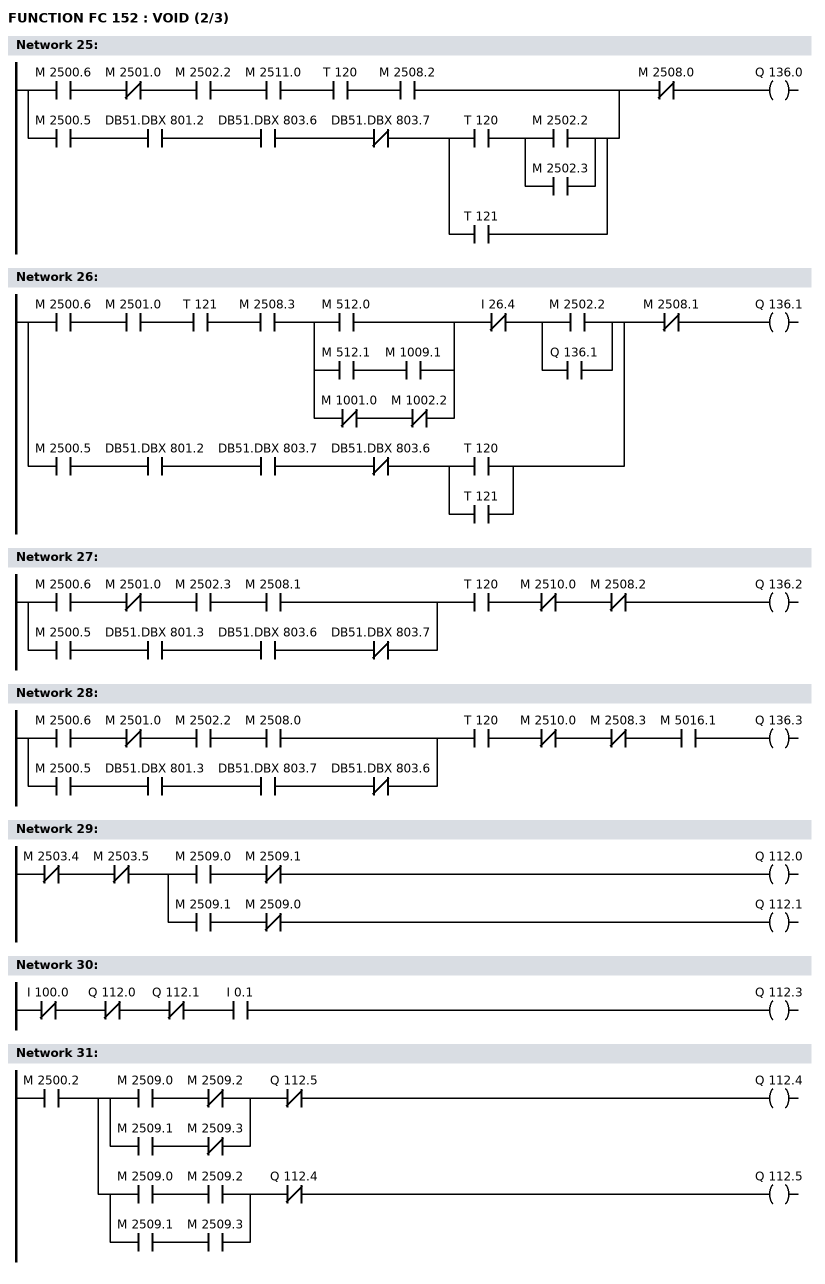

      A(    ;
      A     M   2500.6;
      AN    M   2501.0;
      A     M   2502.2;
      A     M   2511.0;
      A     T    120;
      A     M   2508.2;
      O     ;
      A     M   2500.5;
      A     DB51.DBX  801.2;
      A     DB51.DBX  803.6;
      AN    DB51.DBX  803.7;
      A(    ;
      A     T    120;
      A(    ;
      O     M   2502.2;
      O     M   2502.3;
      )     ;
      O     T    121;
      )     ;
      )     ;
      AN    M   2508.0;
      =     Q    136.0;
NETWORK
TITLE =

      A(    ;
      A     M   2500.6;
      A     M   2501.0;
      A     T    121;
      A     M   2508.3;
      A(    ;
      O     M    512.0;
      O     ;
      A     M    512.1;
      A     M   1009.1;
      O     ;
      AN    M   1001.0;
      AN    M   1002.2;
      )     ;
      AN    I     26.4;
      A(    ;
      O     M   2502.2;
      O     Q    136.1;
      )     ;
      O     ;
      A     M   2500.5;
      A     DB51.DBX  801.2;
      A     DB51.DBX  803.7;
      AN    DB51.DBX  803.6;
      A(    ;
      O     T    120;
      O     T    121;
      )     ;
      )     ;
      AN    M   2508.1;
      =     Q    136.1;
NETWORK
TITLE =

      A(    ;
      A     M   2500.6;
      AN    M   2501.0;
      A     M   2502.3;
      A     M   2508.1;
      O     ;
      A     M   2500.5;
      A     DB51.DBX  801.3;
      A     DB51.DBX  803.6;
      AN    DB51.DBX  803.7;
      )     ;
      A     T    120;
      AN    M   2510.0;
      AN    M   2508.2;
      =     Q    136.2;
NETWORK
TITLE =

      A(    ;
      A     M   2500.6;
      AN    M   2501.0;
      A     M   2502.2;
      A     M   2508.0;
      O     ;
      A     M   2500.5;
      A     DB51.DBX  801.3;
      A     DB51.DBX  803.7;
      AN    DB51.DBX  803.6;
      )     ;
      A     T    120;
      AN    M   2510.0;
      AN    M   2508.3;
      A     M   5016.1;
      =     Q    136.3;
NETWORK
TITLE =

      AN    M   2503.4;
      AN    M   2503.5;
      =     L      0.0;
      A     L      0.0;
      A     M   2509.0;
      AN    M   2509.1;
      =     Q    112.0;
      A     L      0.0;
      A     M   2509.1;
      AN    M   2509.0;
      =     Q    112.1;
NETWORK
TITLE =

      AN    I    100.0;
      AN    Q    112.0;
      AN    Q    112.1;
      A     I      0.1;
      =     Q    112.3;
NETWORK
TITLE =

      A     M   2500.2;
      =     L      0.0;
      A     L      0.0;
      A(    ;
      A     M   2509.0;
      AN    M   2509.2;
      O     ;
      A     M   2509.1;
      AN    M   2509.3;
      )     ;
      AN    Q    112.5;
      =     Q    112.4;
      A     L      0.0;
      A(    ;
      A     M   2509.0;
      A     M   2509.2;
      O     ;
      A     M   2509.1;
      A     M   2509.3;
      )     ;
      AN    Q    112.4;
      =     Q    112.5;
NETWORK
TITLE =
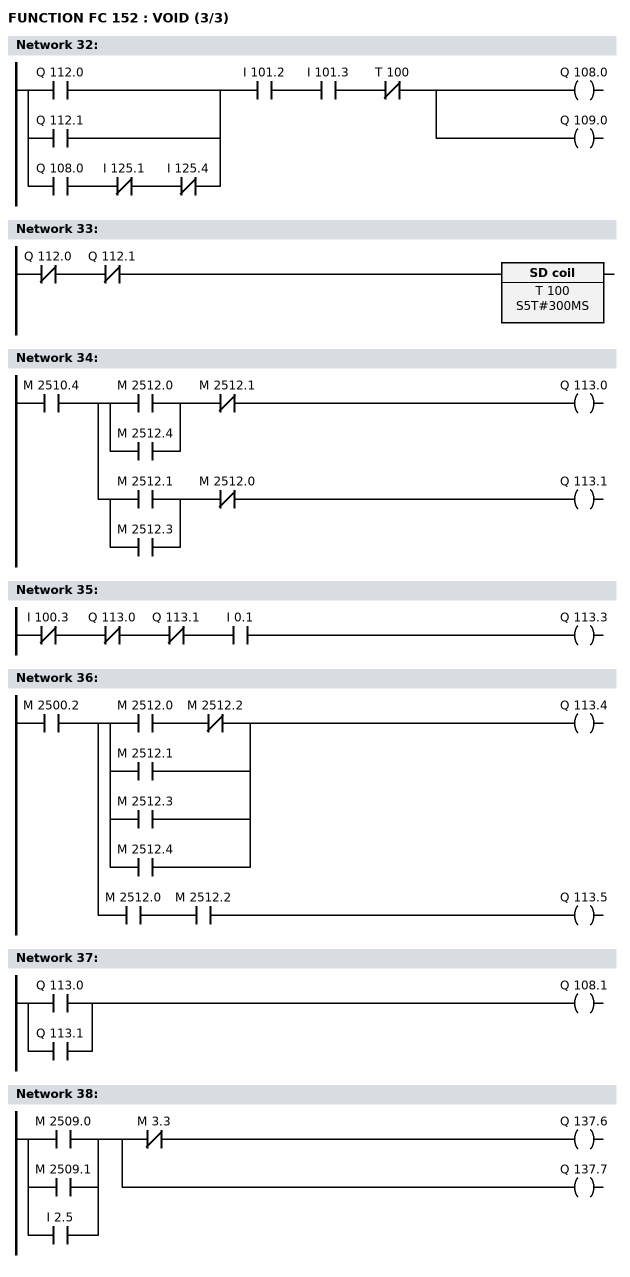

      A(    ;
      O     Q    112.0;
      O     Q    112.1;
      O     ;
      A     Q    108.0;
      AN    I    125.1;
      AN    I    125.4;
      )     ;
      A     I    101.2;
      A     I    101.3;
      AN    T    100;
      =     Q    108.0;
      =     Q    109.0;
NETWORK
TITLE =

      AN    Q    112.0;
      AN    Q    112.1;
      L     S5T#300MS;
      SD    T    100;
NETWORK
TITLE =

      A     M   2510.4;
      =     L      0.0;
      A     L      0.0;
      A(    ;
      O     M   2512.0;
      O     M   2512.4;
      )     ;
      AN    M   2512.1;
      =     Q    113.0;
      A     L      0.0;
      A(    ;
      O     M   2512.1;
      O     M   2512.3;
      )     ;
      AN    M   2512.0;
      =     Q    113.1;
NETWORK
TITLE =

      AN    I    100.3;
      AN    Q    113.0;
      AN    Q    113.1;
      A     I      0.1;
      =     Q    113.3;
NETWORK
TITLE =

      A     M   2500.2;
      =     L      0.0;
      A     L      0.0;
      A(    ;
      A     M   2512.0;
      AN    M   2512.2;
      O     M   2512.1;
      O     M   2512.3;
      O     M   2512.4;
      )     ;
      =     Q    113.4;
      A     L      0.0;
      A     M   2512.0;
      A     M   2512.2;
      =     Q    113.5;
NETWORK
TITLE =

      O     Q    113.0;
      O     Q    113.1;
      =     Q    108.1;
NETWORK
TITLE =

      O     M   2509.0;
      O     M   2509.1;
      O     I      2.5;
      =     L      0.0;
      A     L      0.0;
      AN    M      3.3;
      =     Q    137.6;
      A     L      0.0;
      BLD   102;
      =     Q    137.7;
END_FUNCTION

FUNCTION FC 324 : VOID
TITLE =
VERSION : 0.1

BEGIN
NETWORK
TITLE =DP DIAGNOSTIC FOR DP MASTER SYSTEM(1)

      AN    OV;
      =     L      0.0;
      BLD   103;
      A     OV;
      =     L      0.1;
      BLD   103;
      CALL FC   325 (
           CHECK_ACTIV              := L      0.0,
           EXTERNAL_DP_INTERFACE    := L      0.1,
           DP_MASTERSYSTEM          := 1,
           DATA_FIELD               := P#DB325.DBX0.0 BYTE 50,
           SUM_SLAVES_DIAG          := DB325.DBW   82,
           LIST_SLAVES_NOT_PRESENT  := P#DB325.DBX 50.0 DWORD 4,
           LIST_SLAVES_ERROR        := P#DB325.DBX 66.0 DWORD 4,
           RETVAL                   := DB325.DBW   84,
           BUSY                     := DB325.DBX   90.0);
      NOP   0;
NETWORK
TITLE =#702R1
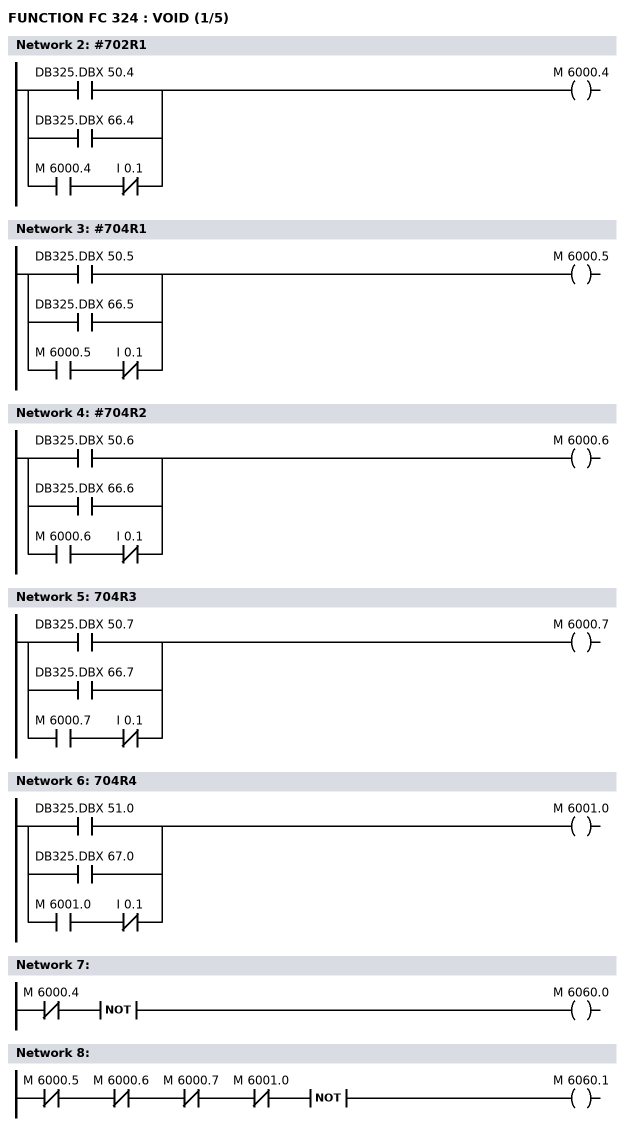

      O     DB325.DBX   50.4;
      O     DB325.DBX   66.4;
      O     ;
      A     M   6000.4;
      AN    I      0.1;
      =     M   6000.4;
NETWORK
TITLE =#704R1

      O     DB325.DBX   50.5;
      O     DB325.DBX   66.5;
      O     ;
      A     M   6000.5;
      AN    I      0.1;
      =     M   6000.5;
NETWORK
TITLE =#704R2

      O     DB325.DBX   50.6;
      O     DB325.DBX   66.6;
      O     ;
      A     M   6000.6;
      AN    I      0.1;
      =     M   6000.6;
NETWORK
TITLE =704R3

      O     DB325.DBX   50.7;
      O     DB325.DBX   66.7;
      O     ;
      A     M   6000.7;
      AN    I      0.1;
      =     M   6000.7;
NETWORK
TITLE =704R4

      O     DB325.DBX   51.0;
      O     DB325.DBX   67.0;
      O     ;
      A     M   6001.0;
      AN    I      0.1;
      =     M   6001.0;
NETWORK
TITLE =

      AN    M   6000.4;
      NOT   ;
      =     M   6060.0;
NETWORK
TITLE =

      AN    M   6000.5;
      AN    M   6000.6;
      AN    M   6000.7;
      AN    M   6001.0;
      NOT   ;
      =     M   6060.1;
NETWORK
TITLE =
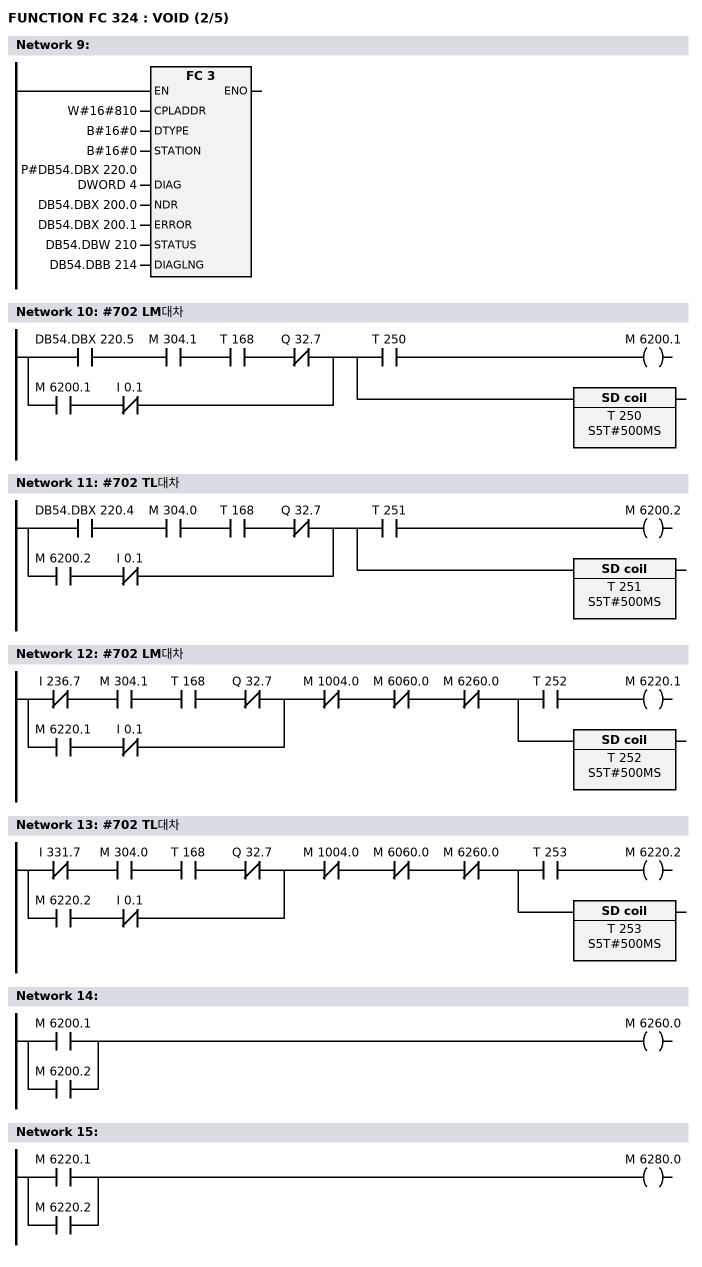

      CALL FC     3 (
           CPLADDR                  := W#16#810,
           DTYPE                    := B#16#0,
           STATION                  := B#16#0,
           DIAG                     := P#DB54.DBX 220.0 DWORD 4,
           NDR                      := DB54.DBX  200.0,
           ERROR                    := DB54.DBX  200.1,
           STATUS                   := DB54.DBW  210,
           DIAGLNG                  := DB54.DBB  214);
      NOP   0;
NETWORK
TITLE =#702 LM대차

      A     DB54.DBX  220.5;
      A     M    304.1;
      A     T    168;
      AN    Q     32.7;
      O     ;
      A     M   6200.1;
      AN    I      0.1;
      =     L      0.0;
      A     L      0.0;
      A     T    250;
      =     M   6200.1;
      A     L      0.0;
      BLD   102;
      L     S5T#500MS;
      SD    T    250;
NETWORK
TITLE =#702 TL대차

      A     DB54.DBX  220.4;
      A     M    304.0;
      A     T    168;
      AN    Q     32.7;
      O     ;
      A     M   6200.2;
      AN    I      0.1;
      =     L      0.0;
      A     L      0.0;
      A     T    251;
      =     M   6200.2;
      A     L      0.0;
      BLD   102;
      L     S5T#500MS;
      SD    T    251;
NETWORK
TITLE =#702 LM대차

      A(    ;
      AN    I    236.7;
      A     M    304.1;
      A     T    168;
      AN    Q     32.7;
      O     ;
      A     M   6220.1;
      AN    I      0.1;
      )     ;
      AN    M   1004.0;
      AN    M   6060.0;
      AN    M   6260.0;
      =     L      0.0;
      A     L      0.0;
      A     T    252;
      =     M   6220.1;
      A     L      0.0;
      BLD   102;
      L     S5T#500MS;
      SD    T    252;
NETWORK
TITLE =#702 TL대차

      A(    ;
      AN    I    331.7;
      A     M    304.0;
      A     T    168;
      AN    Q     32.7;
      O     ;
      A     M   6220.2;
      AN    I      0.1;
      )     ;
      AN    M   1004.0;
      AN    M   6060.0;
      AN    M   6260.0;
      =     L      0.0;
      A     L      0.0;
      A     T    253;
      =     M   6220.2;
      A     L      0.0;
      BLD   102;
      L     S5T#500MS;
      SD    T    253;
NETWORK
TITLE =

      O     M   6200.1;
      O     M   6200.2;
      =     M   6260.0;
NETWORK
TITLE =

      O     M   6220.1;
      O     M   6220.2;
      =     M   6280.0;
NETWORK
TITLE =
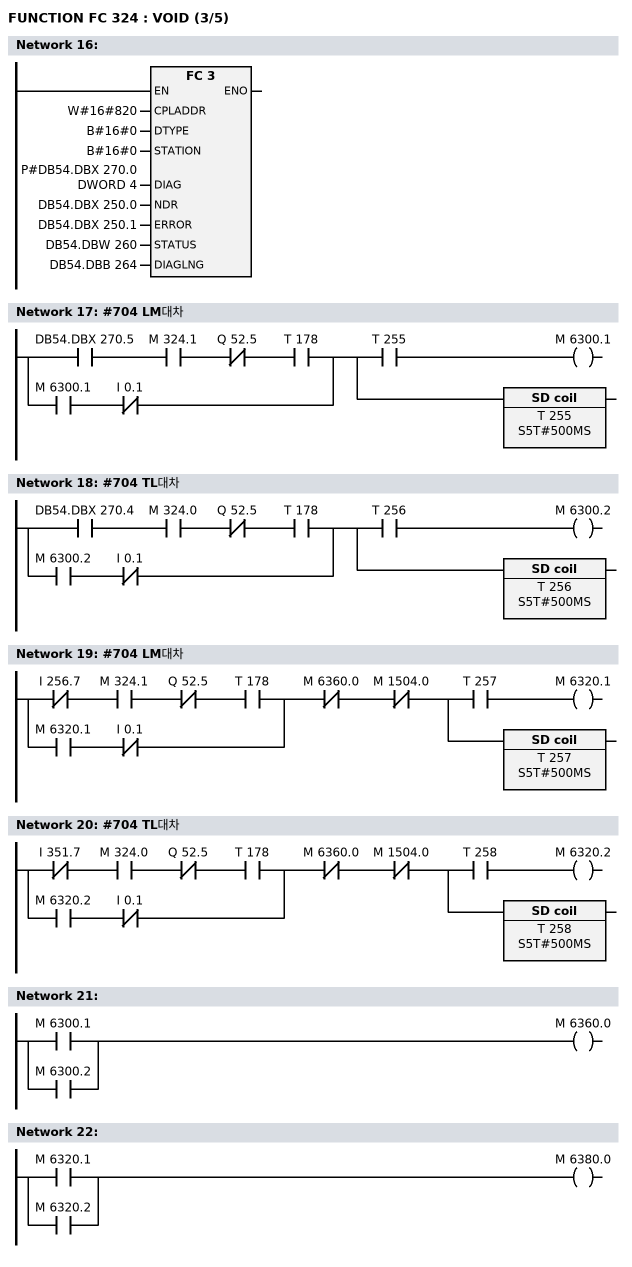

      CALL FC     3 (
           CPLADDR                  := W#16#820,
           DTYPE                    := B#16#0,
           STATION                  := B#16#0,
           DIAG                     := P#DB54.DBX 270.0 DWORD 4,
           NDR                      := DB54.DBX  250.0,
           ERROR                    := DB54.DBX  250.1,
           STATUS                   := DB54.DBW  260,
           DIAGLNG                  := DB54.DBB  264);
      NOP   0;
NETWORK
TITLE =#704 LM대차

      A     DB54.DBX  270.5;
      A     M    324.1;
      AN    Q     52.5;
      A     T    178;
      O     ;
      A     M   6300.1;
      AN    I      0.1;
      =     L      0.0;
      A     L      0.0;
      A     T    255;
      =     M   6300.1;
      A     L      0.0;
      BLD   102;
      L     S5T#500MS;
      SD    T    255;
NETWORK
TITLE =#704 TL대차

      A     DB54.DBX  270.4;
      A     M    324.0;
      AN    Q     52.5;
      A     T    178;
      O     ;
      A     M   6300.2;
      AN    I      0.1;
      =     L      0.0;
      A     L      0.0;
      A     T    256;
      =     M   6300.2;
      A     L      0.0;
      BLD   102;
      L     S5T#500MS;
      SD    T    256;
NETWORK
TITLE =#704 LM대차

      A(    ;
      AN    I    256.7;
      A     M    324.1;
      AN    Q     52.5;
      A     T    178;
      O     ;
      A     M   6320.1;
      AN    I      0.1;
      )     ;
      AN    M   6360.0;
      AN    M   1504.0;
      =     L      0.0;
      A     L      0.0;
      A     T    257;
      =     M   6320.1;
      A     L      0.0;
      BLD   102;
      L     S5T#500MS;
      SD    T    257;
NETWORK
TITLE =#704 TL대차

      A(    ;
      AN    I    351.7;
      A     M    324.0;
      AN    Q     52.5;
      A     T    178;
      O     ;
      A     M   6320.2;
      AN    I      0.1;
      )     ;
      AN    M   6360.0;
      AN    M   1504.0;
      =     L      0.0;
      A     L      0.0;
      A     T    258;
      =     M   6320.2;
      A     L      0.0;
      BLD   102;
      L     S5T#500MS;
      SD    T    258;
NETWORK
TITLE =

      O     M   6300.1;
      O     M   6300.2;
      =     M   6360.0;
NETWORK
TITLE =

      O     M   6320.1;
      O     M   6320.2;
      =     M   6380.0;
NETWORK
TITLE =
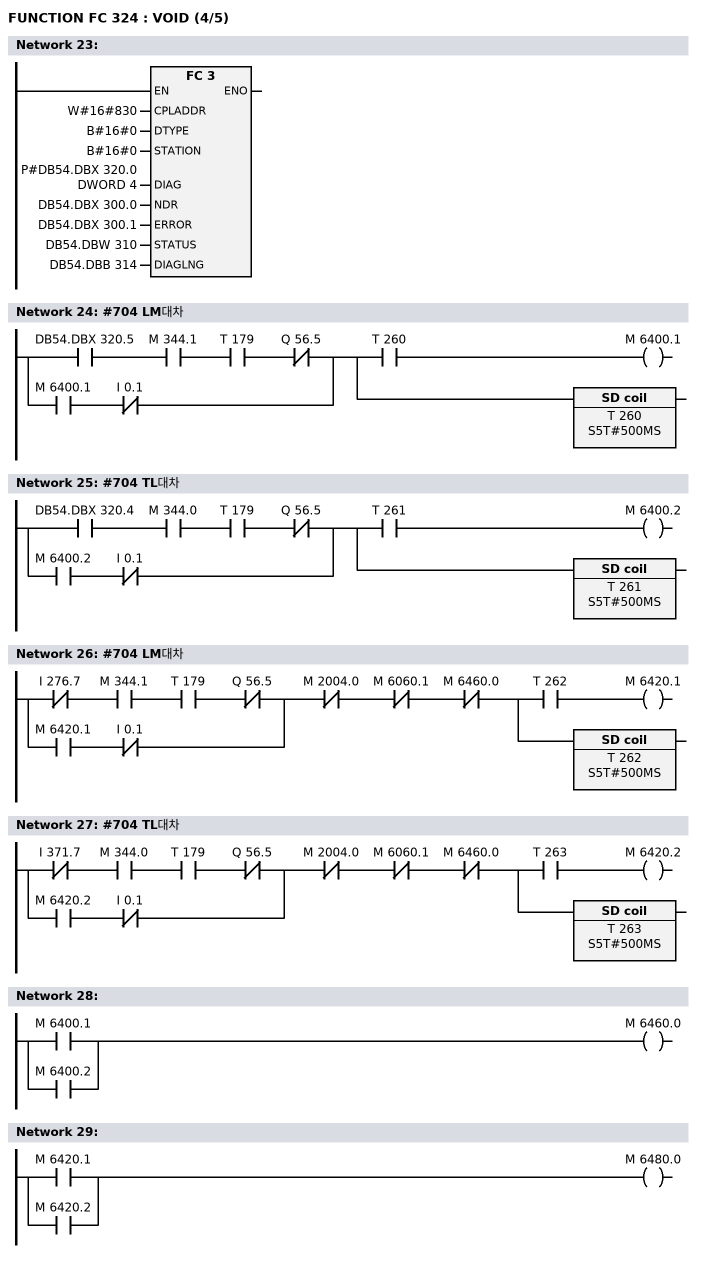

      CALL FC     3 (
           CPLADDR                  := W#16#830,
           DTYPE                    := B#16#0,
           STATION                  := B#16#0,
           DIAG                     := P#DB54.DBX 320.0 DWORD 4,
           NDR                      := DB54.DBX  300.0,
           ERROR                    := DB54.DBX  300.1,
           STATUS                   := DB54.DBW  310,
           DIAGLNG                  := DB54.DBB  314);
      NOP   0;
NETWORK
TITLE =#704 LM대차

      A     DB54.DBX  320.5;
      A     M    344.1;
      A     T    179;
      AN    Q     56.5;
      O     ;
      A     M   6400.1;
      AN    I      0.1;
      =     L      0.0;
      A     L      0.0;
      A     T    260;
      =     M   6400.1;
      A     L      0.0;
      BLD   102;
      L     S5T#500MS;
      SD    T    260;
NETWORK
TITLE =#704 TL대차

      A     DB54.DBX  320.4;
      A     M    344.0;
      A     T    179;
      AN    Q     56.5;
      O     ;
      A     M   6400.2;
      AN    I      0.1;
      =     L      0.0;
      A     L      0.0;
      A     T    261;
      =     M   6400.2;
      A     L      0.0;
      BLD   102;
      L     S5T#500MS;
      SD    T    261;
NETWORK
TITLE =#704 LM대차

      A(    ;
      AN    I    276.7;
      A     M    344.1;
      A     T    179;
      AN    Q     56.5;
      O     ;
      A     M   6420.1;
      AN    I      0.1;
      )     ;
      AN    M   2004.0;
      AN    M   6060.1;
      AN    M   6460.0;
      =     L      0.0;
      A     L      0.0;
      A     T    262;
      =     M   6420.1;
      A     L      0.0;
      BLD   102;
      L     S5T#500MS;
      SD    T    262;
NETWORK
TITLE =#704 TL대차

      A(    ;
      AN    I    371.7;
      A     M    344.0;
      A     T    179;
      AN    Q     56.5;
      O     ;
      A     M   6420.2;
      AN    I      0.1;
      )     ;
      AN    M   2004.0;
      AN    M   6060.1;
      AN    M   6460.0;
      =     L      0.0;
      A     L      0.0;
      A     T    263;
      =     M   6420.2;
      A     L      0.0;
      BLD   102;
      L     S5T#500MS;
      SD    T    263;
NETWORK
TITLE =

      O     M   6400.1;
      O     M   6400.2;
      =     M   6460.0;
NETWORK
TITLE =

      O     M   6420.1;
      O     M   6420.2;
      =     M   6480.0;
NETWORK
TITLE =
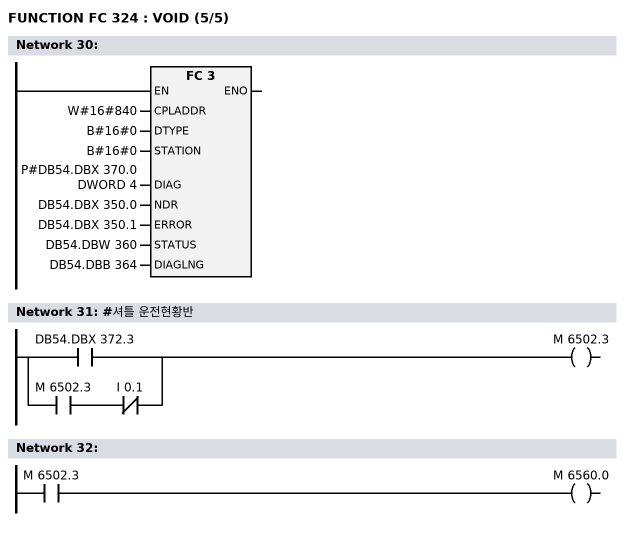

      CALL FC     3 (
           CPLADDR                  := W#16#840,
           DTYPE                    := B#16#0,
           STATION                  := B#16#0,
           DIAG                     := P#DB54.DBX 370.0 DWORD 4,
           NDR                      := DB54.DBX  350.0,
           ERROR                    := DB54.DBX  350.1,
           STATUS                   := DB54.DBW  360,
           DIAGLNG                  := DB54.DBB  364);
      NOP   0;
NETWORK
TITLE =#셔틀 운전현황반

      O     DB54.DBX  372.3;
      O     ;
      A     M   6502.3;
      AN    I      0.1;
      =     M   6502.3;
NETWORK
TITLE =

      A     M   6502.3;
      =     M   6560.0;
END_FUNCTION

FUNCTION FC 501 : VOID
TITLE =
VERSION : 0.1


VAR_INPUT
  IN0 : INT ;
  IN1 : INT ;
  IN2 : INT ;
  IN3 : INT ;
  IN4 : INT ;
  IN5 : INT ;
  IN6 : INT ;
  IN7 : BOOL ;
  IN8 : BOOL ;
  IN9 : BOOL ;
  IN10 : BOOL ;
  IN11 : BOOL ;
  IN12 : BOOL ;
END_VAR
VAR_OUTPUT
  OUT13 : BOOL ;
  OUT14 : BOOL ;
END_VAR
VAR_TEMP
  TEMP15 : INT ;
  TEMP16 : INT ;
  TEMP17 : INT ;
  TEMP18 : INT ;
  TEMP19 : INT ;
  TEMP20 : INT ;
  TEMP21 : INT ;
  TEMP22 : BOOL ;
  TEMP23 : WORD ;
  TEMP24 : WORD ;
  TEMP25 : INT ;
  TEMP26 : WORD ;
  TEMP27 : INT ;
  TEMP28 : INT ;
  TEMP29 : INT ;
  TEMP30 : INT ;
END_VAR
BEGIN
NETWORK
TITLE =

      L     #IN0;
      T     #TEMP15;
      L     #IN1;
      T     #TEMP16;
      L     #IN2;
      T     #TEMP17;
      L     #IN3;
      T     #TEMP18;
      OPN   DI [#TEMP17];
NETWORK
TITLE =

      CALL FC   504 (
           IN0                      := #TEMP18,
           IN1                      := #IN4,
           IN2                      := 16,
           IN3                      := #TEMP17,
           IN4                      := 16);
      NOP   0;
NETWORK
TITLE =

      A(    ;
      L     DIW   17;
      L     DIW   18;
      OW    ;
      T     #TEMP24;
      SET   ;
      SAVE  ;
      CLR   ;
      A     BR;
      )     ;
      JNB   M001;
      L     DIW   18;
      T     #TEMP24;
M001: NOP   0;
NETWORK
TITLE =

      A(    ;
      L     60;
      L     #TEMP15;
      *I    ;
      T     #TEMP20;
      AN    OV;
      SAVE  ;
      CLR   ;
      A     BR;
      )     ;
      JNB   M002;
      L     #TEMP20;
      L     60;
      -I    ;
      T     #TEMP21;
M002: NOP   0;
NETWORK
TITLE =

      O(    ;
      L     0;
      L     #TEMP15;
      ==I   ;
      )     ;
      O(    ;
      L     16;
      L     #TEMP15;
      <I    ;
      )     ;
      SAVE  ;
      BEC   ;
NETWORK
TITLE =

      OPN   DB [#TEMP16];
      L     #TEMP21;
      SLW   3;
      LAR1  ;
NETWORK
TITLE =
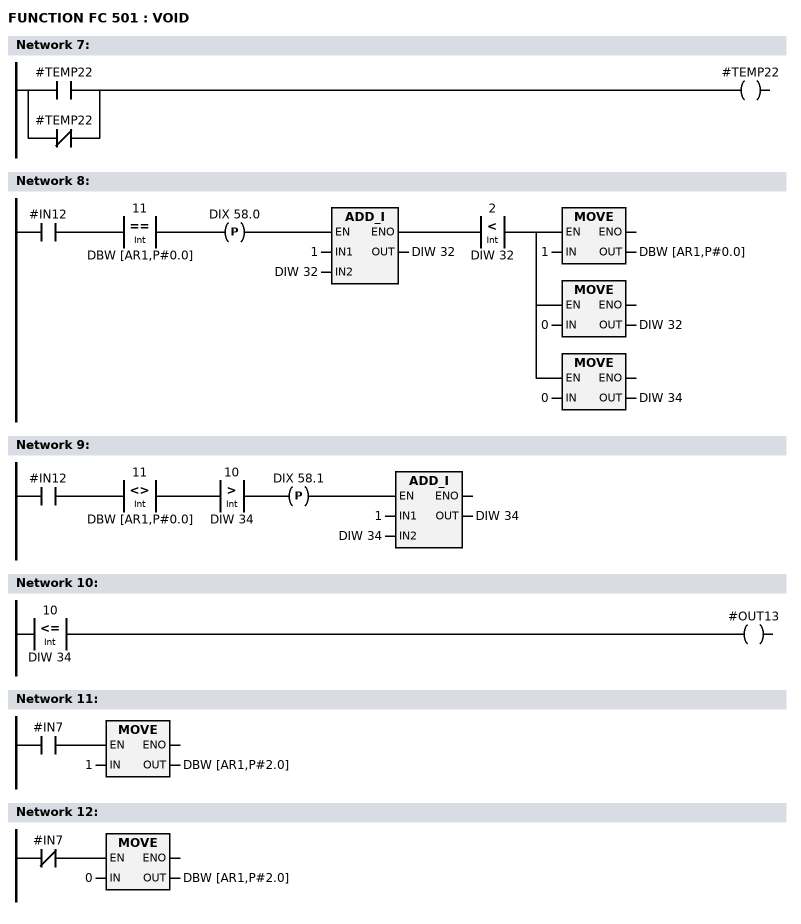

      O     #TEMP22;
      ON    #TEMP22;
      =     #TEMP22;
NETWORK
TITLE =

      A(    ;
      A     #IN12;
      A(    ;
      L     11;
      L     DBW [AR1,P#0.0];
      ==I   ;
      )     ;
      FP    DIX   58.0;
      JNB   M003;
      L     1;
      L     DIW   32;
      +I    ;
      T     DIW   32;
      AN    OV;
      SAVE  ;
      CLR   ;
M003: A     BR;
      )     ;
      A(    ;
      L     2;
      L     DIW   32;
      <I    ;
      )     ;
      =     L     32.0;
      A     L     32.0;
      JNB   M005;
      L     1;
      T     DBW [AR1,P#0.0];
M005: NOP   0;
      A     L     32.0;
      JNB   M006;
      L     0;
      T     DIW   32;
M006: NOP   0;
      A     L     32.0;
      JNB   M007;
      L     0;
      T     DIW   34;
M007: NOP   0;
NETWORK
TITLE =

      A     #IN12;
      A(    ;
      L     11;
      L     DBW [AR1,P#0.0];
      <>I   ;
      )     ;
      A(    ;
      L     10;
      L     DIW   34;
      >I    ;
      )     ;
      FP    DIX   58.1;
      JNB   M004;
      L     1;
      L     DIW   34;
      +I    ;
      T     DIW   34;
M004: NOP   0;
NETWORK
TITLE =

      L     10;
      L     DIW   34;
      <=I   ;
      =     #OUT13;
NETWORK
TITLE =

      A     #IN7;
      JNB   M008;
      L     1;
      T     DBW [AR1,P#2.0];
M008: NOP   0;
NETWORK
TITLE =

      AN    #IN7;
      JNB   M009;
      L     0;
      T     DBW [AR1,P#2.0];
M009: NOP   0;
NETWORK
TITLE =

      L     #TEMP21;
      SLW   3;
      LAR1  ;
      A     #IN8;
      FP    DIX   58.2;
      JNB   M00a;
      L     1;
      T     DBW [AR1,P#4.0];
M00a: NOP   0;
NETWORK
TITLE =

      L     #TEMP21;
      SLW   3;
      LAR1  ;
      A(    ;
      A     #IN8;
      FN    DIX   58.3;
      JNB   M00b;
      L     0;
      T     DBW [AR1,P#4.0];
      SET   ;
      SAVE  ;
      CLR   ;
M00b: A     BR;
      )     ;
      JNB   M00c;
      L     0;
      T     DBW [AR1,P#6.0];
M00c: NOP   0;
NETWORK
TITLE =

      L     #TEMP21;
      SLW   3;
      LAR1  ;
      A(    ;
      L     1;
      L     DBW [AR1,P#4.0];
      ==I   ;
      )     ;
      FP    DIX   58.4;
      JNB   M00d;
      CALL FC   502 (
           IN0                      := #TEMP17,
           IN1                      := W#16#400,
           IN2                      := 0,
           IN3                      := #TEMP24);
M00d: NOP   0;
NETWORK
TITLE =

      L     #TEMP21;
      SLW   3;
      LAR1  ;
      A(    ;
      L     0;
      L     DBW [AR1,P#4.0];
      ==I   ;
      )     ;
      FP    DIX   58.5;
      JNB   M00e;
      CALL FC   502 (
           IN0                      := #TEMP17,
           IN1                      := W#16#500,
           IN2                      := 0,
           IN3                      := #TEMP24);
M00e: NOP   0;
NETWORK
TITLE =

      L     #TEMP21;
      SLW   3;
      LAR1  ;
      A(    ;
      A     #IN9;
      AN    DIX   61.0;
      FP    DIX   58.6;
      JNB   M00f;
      L     1;
      T     DBW [AR1,P#22.0];
      SET   ;
      SAVE  ;
      CLR   ;
M00f: A     BR;
      )     ;
      JNB   M010;
      L     1;
      L     DBW [AR1,P#6.0];
      +I    ;
      T     DBW [AR1,P#6.0];
M010: NOP   0;
NETWORK
TITLE =

      L     #TEMP21;
      SLW   3;
      LAR1  ;
      A(    ;
      L     1;
      L     DBW [AR1,P#22.0];
      ==I   ;
      )     ;
      FP    DIX   60.1;
      =     L     32.0;
      A(    ;
      A     L     32.0;
      JNB   M011;
      L     40;
      L     #TEMP21;
      +I    ;
      T     #TEMP29;
      AN    OV;
      SAVE  ;
      CLR   ;
M011: A     BR;
      )     ;
      JNB   M015;
      CALL FC   504 (
           IN0                      := #TEMP16,
           IN1                      := #TEMP29,
           IN2                      := 16,
           IN3                      := #TEMP17,
           IN4                      := 0);
M015: NOP   0;
      A(    ;
      A     L     32.0;
      JNB   M016;
      L     24;
      L     #TEMP21;
      +I    ;
      T     #TEMP28;
      AN    OV;
      SAVE  ;
      CLR   ;
M016: A     BR;
      )     ;
      JNB   M017;
      CALL FC   503 (
           IN0                      := #TEMP16,
           IN1                      := 16,
           IN2                      := #TEMP28,
           IN3                      := B#16#0);
M017: NOP   0;
      A(    ;
      A     L     32.0;
      JNB   M018;
      L     40;
      L     #TEMP21;
      +I    ;
      T     #TEMP28;
      AN    OV;
      SAVE  ;
      CLR   ;
M018: A     BR;
      )     ;
      JNB   M019;
      CALL FC   503 (
           IN0                      := #TEMP16,
           IN1                      := 16,
           IN2                      := #TEMP28,
           IN3                      := B#16#0);
M019: NOP   0;
NETWORK
TITLE =

      L     #TEMP21;
      SLW   3;
      LAR1  ;
      A(    ;
      L     DBW [AR1,P#6.0];
      T     #TEMP27;
      SET   ;
      SAVE  ;
      CLR   ;
      A     BR;
      )     ;
      JNB   M01a;
      L     DBW [AR1,P#8.0];
      T     #TEMP26;
M01a: NOP   0;
NETWORK
TITLE =

      L     #TEMP21;
      SLW   3;
      LAR1  ;
      A(    ;
      L     1;
      L     DBW [AR1,P#22.0];
      ==I   ;
      )     ;
      FP    DIX   58.7;
      JNB   M01b;
      CALL FC   502 (
           IN0                      := #TEMP17,
           IN1                      := W#16#200,
           IN2                      := #TEMP27,
           IN3                      := #TEMP26);
M01b: NOP   0;
NETWORK
TITLE =

      L     DBW [AR1,P#22.0];
      T     #TEMP25;
      NOP   0;
NETWORK
TITLE =

      L     DBW [AR1,P#24.0];
      T     #TEMP23;
      NOP   0;
NETWORK
TITLE =

      L     #TEMP21;
      SLW   3;
      LAR1  ;
      A(    ;
      L     0;
      L     DBW [AR1,P#22.0];
      <>I   ;
      )     ;
      A(    ;
      L     1;
      L     DBW [AR1,P#22.0];
      <>I   ;
      )     ;
      A(    ;
      L     DIW   36;
      L     DBW [AR1,P#22.0];
      <>I   ;
      )     ;
      FP    DIX   59.0;
      =     L     32.0;
      A     L     32.0;
      A(    ;
      L     99;
      L     DBW [AR1,P#22.0];
      <>I   ;
      )     ;
      A(    ;
      L     100;
      L     DBW [AR1,P#22.0];
      <>I   ;
      )     ;
      JNB   M01c;
      CALL FC   502 (
           IN0                      := #TEMP17,
           IN1                      := W#16#300,
           IN2                      := #TEMP25,
           IN3                      := #TEMP23);
M01c: NOP   0;
      A     L     32.0;
      AN    #TEMP22;
      A(    ;
      L     99;
      L     DBW [AR1,P#22.0];
      ==I   ;
      )     ;
      JNB   M01d;
      CALL FC   502 (
           IN0                      := #TEMP17,
           IN1                      := W#16#700,
           IN2                      := #TEMP25,
           IN3                      := #TEMP23);
M01d: NOP   0;
      A     L     32.0;
      A(    ;
      L     100;
      L     DBW [AR1,P#22.0];
      ==I   ;
      )     ;
      JNB   M01e;
      CALL FC   502 (
           IN0                      := #TEMP17,
           IN1                      := W#16#600,
           IN2                      := #TEMP25,
           IN3                      := #TEMP23);
M01e: NOP   0;
      A     L     32.0;
      BLD   102;
      R     DIX   52.2;
      A     L     32.0;
      BLD   102;
      R     DIX   52.3;
NETWORK
TITLE =

      L     #TEMP21;
      SLW   3;
      LAR1  ;
      A(    ;
      A(    ;
      L     100;
      L     DBW [AR1,P#22.0];
      ==I   ;
      )     ;
      FP    DIX   59.1;
      JNB   M01f;
      L     0;
      T     DBW [AR1,P#6.0];
      SET   ;
      SAVE  ;
      CLR   ;
M01f: A     BR;
      )     ;
      JNB   M020;
      CALL FC   503 (
           IN0                      := #TEMP17,
           IN1                      := 16,
           IN2                      := 0,
           IN3                      := B#16#0);
M020: A     BR;
      S     DIX   61.0;
NETWORK
TITLE =

      A     #IN8;
      FN    DIX   61.1;
      R     DIX   61.0;
NETWORK
TITLE =

      L     #TEMP21;
      SLW   3;
      LAR1  ;
      A(    ;
      O(    ;
      L     11;
      L     DBW [AR1,P#22.0];
      ==I   ;
      )     ;
      O(    ;
      L     99;
      L     DBW [AR1,P#22.0];
      ==I   ;
      )     ;
      )     ;
      FP    DIX   59.2;
      A(    ;
      L     L#0;
      L     DID    0;
      <>D   ;
      )     ;
      =     L     32.0;
      A     L     32.0;
      A(    ;
      L     DBD [AR1,P#24.0];
      L     DBD [AR1,P#8.0];
      <>D   ;
      )     ;
      S     DIX   52.0;
      A     L     32.0;
      A(    ;
      L     DBD [AR1,P#24.0];
      L     DID    0;
      ==D   ;
      )     ;
      A(    ;
      L     DBD [AR1,P#28.0];
      L     DID    4;
      ==D   ;
      )     ;
      A(    ;
      L     DBD [AR1,P#32.0];
      L     DID    8;
      ==D   ;
      )     ;
      A(    ;
      L     DBD [AR1,P#36.0];
      L     DID   12;
      ==D   ;
      )     ;
      S     DIX   52.1;
      A     L     32.0;
      BLD   102;
      S     DIX   61.2;
NETWORK
TITLE =

      L     #TEMP21;
      SLW   3;
      LAR1  ;
      A(    ;
      O(    ;
      L     11;
      L     DBW [AR1,P#22.0];
      ==I   ;
      )     ;
      O(    ;
      L     99;
      L     DBW [AR1,P#22.0];
      ==I   ;
      )     ;
      )     ;
      A     DIX   52.0;
      A     DIX   52.1;
      O(    ;
      L     100;
      L     DBW [AR1,P#22.0];
      ==I   ;
      )     ;
      O(    ;
      L     0;
      L     #TEMP19;
      ==I   ;
      )     ;
      O     ;
      A(    ;
      L     L#0;
      L     DID    0;
      ==D   ;
      )     ;
      A(    ;
      L     L#0;
      L     DID    4;
      ==D   ;
      )     ;
      S     DIX   52.2;
NETWORK
TITLE =

      L     #TEMP21;
      SLW   3;
      LAR1  ;
      A(    ;
      O(    ;
      L     11;
      L     DBW [AR1,P#22.0];
      ==I   ;
      )     ;
      O(    ;
      L     99;
      L     DBW [AR1,P#22.0];
      ==I   ;
      )     ;
      )     ;
      A(    ;
      ON    DIX   52.0;
      ON    DIX   52.1;
      )     ;
      A(    ;
      L     L#0;
      L     DBD [AR1,P#24.0];
      <>D   ;
      )     ;
      A     DIX   61.2;
      A(    ;
      L     0;
      L     #IN5;
      <>I   ;
      )     ;
      A(    ;
      L     L#0;
      L     DID    0;
      <>D   ;
      )     ;
      A(    ;
      L     L#0;
      L     DID    4;
      <>D   ;
      )     ;
      S     DIX   52.3;
NETWORK
TITLE =

      L     #TEMP21;
      SLW   3;
      LAR1  ;
      A(    ;
      L     99;
      L     DBW [AR1,P#22.0];
      ==I   ;
      )     ;
      FP    DIX   59.3;
      S     DIX   52.6;
NETWORK
TITLE =

      L     #TEMP21;
      SLW   3;
      LAR1  ;
      A     DIX   52.6;
      A(    ;
      O(    ;
      L     11;
      L     DBW [AR1,P#22.0];
      ==I   ;
      )     ;
      O(    ;
      L     100;
      L     DBW [AR1,P#22.0];
      ==I   ;
      )     ;
      )     ;
      R     DIX   52.6;
NETWORK
TITLE =

      L     #TEMP21;
      SLW   3;
      LAR1  ;
      AN    DIX   52.2;
      A     DIX   52.3;
      A(    ;
      L     0;
      L     #TEMP19;
      <>I   ;
      )     ;
      FP    DIX   59.5;
      =     L     32.0;
      A     L     32.0;
      AN    DIX   52.0;
      JNB   M021;
      L     1;
      T     DBW [AR1,P#12.0];
M021: NOP   0;
      A     L     32.0;
      A     DIX   52.0;
      AN    DIX   52.1;
      JNB   M022;
      L     2;
      T     DBW [AR1,P#12.0];
M022: NOP   0;
NETWORK
TITLE =

      L     #TEMP21;
      SLW   3;
      LAR1  ;
      A(    ;
      A(    ;
      O     DIX   52.2;
      O     DIX   52.3;
      )     ;
      A(    ;
      L     1;
      L     DBW [AR1,P#22.0];
      <>I   ;
      )     ;
      A(    ;
      L     3;
      L     DBW [AR1,P#22.0];
      <>I   ;
      )     ;
      FP    DIX   59.4;
      JNB   M023;
      L     3;
      T     DBW [AR1,P#22.0];
      SET   ;
      SAVE  ;
      CLR   ;
M023: A     BR;
      )     ;
      JNB   M024;
      L     DBW [AR1,P#22.0];
      T     DIW   36;
      SET   ;
      SAVE  ;
      CLR   ;
M024: A     BR;
      R     DIX   52.0;
      R     DIX   52.1;
      R     DIX   61.2;
NETWORK
TITLE =

      AN    DIX   52.2;
      A     DIX   52.3;
      O     DIX   52.6;
      =     #OUT14;
NETWORK
TITLE =

      L     #TEMP21;
      SLW   3;
      LAR1  ;
      A(    ;
      L     3;
      L     DBW [AR1,P#22.0];
      ==I   ;
      )     ;
      A     DIX   52.2;
      =     L     32.0;
      A     L     32.0;
      BLD   102;
      =     DIX   52.7;
      A     L     32.0;
      JNB   M025;
      L     0;
      T     DBW [AR1,P#12.0];
M025: NOP   0;
NETWORK
TITLE =

      L     #TEMP21;
      SLW   3;
      LAR1  ;
      A(    ;
      L     DBW [AR1,P#24.0];
      T     DIW 1102;
      SET   ;
      SAVE  ;
      CLR   ;
      A     BR;
      )     ;
      JNB   M026;
      L     DBW [AR1,P#26.0];
      T     DIW 1100;
M026: NOP   0;
NETWORK
TITLE =

      L     #TEMP21;
      SLW   3;
      LAR1  ;
      A(    ;
      A(    ;
      A(    ;
      L     DBB [AR1,P#28.0];
      T     DIB 1105;
      SET   ;
      SAVE  ;
      CLR   ;
      A     BR;
      )     ;
      JNB   M027;
      L     DBB [AR1,P#29.0];
      T     DIB 1104;
      SET   ;
      SAVE  ;
      CLR   ;
M027: A     BR;
      )     ;
      JNB   M012;
      L     DBB [AR1,P#30.0];
      T     DIB 1107;
      SET   ;
      SAVE  ;
      CLR   ;
M012: A     BR;
      )     ;
      JNB   M013;
      L     DBB [AR1,P#31.0];
      T     DIB 1106;
M013: NOP   0;
NETWORK
TITLE =

      L     #TEMP21;
      SLW   3;
      LAR1  ;
      A(    ;
      A(    ;
      A(    ;
      L     DBB [AR1,P#32.0];
      T     DIB 1109;
      SET   ;
      SAVE  ;
      CLR   ;
      A     BR;
      )     ;
      JNB   M014;
      L     DBB [AR1,P#33.0];
      T     DIB 1108;
      SET   ;
      SAVE  ;
      CLR   ;
M014: A     BR;
      )     ;
      JNB   M028;
      L     DBB [AR1,P#34.0];
      T     DIB 1111;
      SET   ;
      SAVE  ;
      CLR   ;
M028: A     BR;
      )     ;
      JNB   M029;
      L     DBB [AR1,P#35.0];
      T     DIB 1110;
M029: NOP   0;
NETWORK
TITLE =

      L     #TEMP21;
      SLW   3;
      LAR1  ;
      A(    ;
      A(    ;
      A(    ;
      L     DBB [AR1,P#36.0];
      T     DIB 1113;
      SET   ;
      SAVE  ;
      CLR   ;
      A     BR;
      )     ;
      JNB   M02a;
      L     DBB [AR1,P#37.0];
      T     DIB 1112;
      SET   ;
      SAVE  ;
      CLR   ;
M02a: A     BR;
      )     ;
      JNB   M02b;
      L     DBB [AR1,P#38.0];
      T     DIB 1115;
      SET   ;
      SAVE  ;
      CLR   ;
M02b: A     BR;
      )     ;
      JNB   M02c;
      L     DBB [AR1,P#39.0];
      T     DIB 1114;
M02c: NOP   0;
NETWORK
TITLE =

      L     #TEMP21;
      SLW   3;
      LAR1  ;
      A(    ;
      A     #IN12;
      A     #IN10;
      FP    DIX   61.3;
      JNB   M03d;
      L     1;
      L     DIW   38;
      +I    ;
      T     DIW   38;
      AN    OV;
      SAVE  ;
      CLR   ;
M03d: A     BR;
      )     ;
      A(    ;
      L     2;
      L     DIW   38;
      <I    ;
      )     ;
      S     DIX   61.4;
NETWORK
TITLE =

      L     #TEMP21;
      SLW   3;
      LAR1  ;
      AN    #IN10;
      JNB   M03e;
      L     0;
      T     DIW   38;
      SET   ;
      SAVE  ;
      CLR   ;
M03e: A     BR;
      R     DIX   61.4;
NETWORK
TITLE =

      L     #TEMP21;
      SLW   3;
      LAR1  ;
      A(    ;
      L     1;
      L     DBW [AR1,P#2.0];
      ==I   ;
      )     ;
      A(    ;
      L     3;
      L     DBW [AR1,P#22.0];
      ==I   ;
      )     ;
      A     #IN10;
      A     DIX   52.7;
      A     DIX   61.4;
      =     L     32.0;
      A     L     32.0;
      JNB   M02d;
      CALL FC   504 (
           IN0                      := #TEMP17,
           IN1                      := 1100,
           IN2                      := 16,
           IN3                      := #IN5,
           IN4                      := #IN6);
M02d: NOP   0;
      A(    ;
      A(    ;
      A     L     32.0;
      JNB   M02e;
      L     24;
      L     #TEMP21;
      +I    ;
      T     #TEMP29;
      AN    OV;
      SAVE  ;
      CLR   ;
M02e: A     BR;
      )     ;
      JNB   M02f;
      L     8;
      L     #TEMP21;
      +I    ;
      T     #TEMP30;
      AN    OV;
      SAVE  ;
      CLR   ;
M02f: A     BR;
      )     ;
      JNB   M030;
      CALL FC   504 (
           IN0                      := #TEMP16,
           IN1                      := #TEMP29,
           IN2                      := 4,
           IN3                      := #TEMP16,
           IN4                      := #TEMP30);
M030: NOP   0;
      A(    ;
      A     L     32.0;
      JNB   M031;
      L     40;
      L     #TEMP21;
      +I    ;
      T     #TEMP29;
      AN    OV;
      SAVE  ;
      CLR   ;
M031: A     BR;
      )     ;
      JNB   M032;
      CALL FC   504 (
           IN0                      := #TEMP16,
           IN1                      := #TEMP29,
           IN2                      := 16,
           IN3                      := #TEMP17,
           IN4                      := 0);
M032: NOP   0;
NETWORK
TITLE =

      L     #TEMP21;
      SLW   3;
      LAR1  ;
      A     #IN11;
      A(    ;
      O     DIX   27.2;
      O     DIX   27.3;
      O     DIX   27.4;
      O     DIX   27.5;
      O     DIX   27.6;
      O     DIX   27.7;
      )     ;
      =     DIX   54.0;
      S     DIX   54.1;
NETWORK
TITLE =
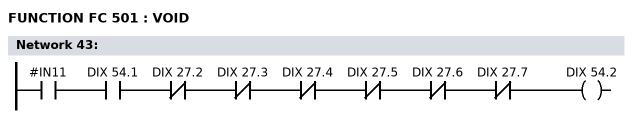

      A     #IN11;
      A     DIX   54.1;
      AN    DIX   27.2;
      AN    DIX   27.3;
      AN    DIX   27.4;
      AN    DIX   27.5;
      AN    DIX   27.6;
      AN    DIX   27.7;
      =     DIX   54.2;
NETWORK
TITLE =

      L     #TEMP21;
      SLW   3;
      LAR1  ;
      A(    ;
      A(    ;
      A(    ;
      A(    ;
      A(    ;
      O     DIX   54.0;
      O     DIX   54.2;
      )     ;
      A(    ;
      L     1;
      L     DBW [AR1,P#22.0];
      <>I   ;
      )     ;
      FP    DIX   59.6;
      JNB   M03f;
      L     1;
      T     DBW [AR1,P#20.0];
      SET   ;
      SAVE  ;
      CLR   ;
M03f: A     BR;
      )     ;
      JNB   M040;
      CALL FC   503 (
           IN0                      := #TEMP17,
           IN1                      := 16,
           IN2                      := 0,
           IN3                      := B#16#0);
M040: A     BR;
      )     ;
      JNB   M041;
      L     24;
      L     #TEMP21;
      +I    ;
      T     #TEMP28;
      AN    OV;
      SAVE  ;
      CLR   ;
M041: A     BR;
      )     ;
      JNB   M042;
      CALL FC   503 (
           IN0                      := #TEMP16,
           IN1                      := 32,
           IN2                      := #TEMP28,
           IN3                      := B#16#0);
M042: A     BR;
      )     ;
      JNB   M043;
      L     0;
      T     DBW [AR1,P#12.0];
      SET   ;
      SAVE  ;
      CLR   ;
M043: NOP   0;
NETWORK
TITLE =
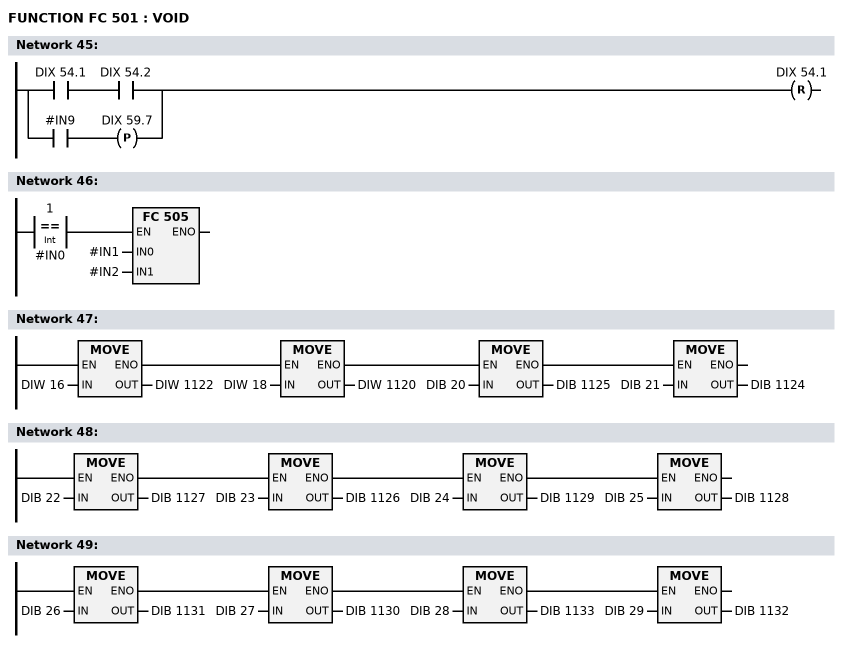

      A     DIX   54.1;
      A     DIX   54.2;
      O(    ;
      A     #IN9;
      FP    DIX   59.7;
      )     ;
      R     DIX   54.1;
NETWORK
TITLE =

      A(    ;
      L     1;
      L     #IN0;
      ==I   ;
      )     ;
      JNB   M033;
      CALL FC   505 (
           IN0                      := #IN1,
           IN1                      := #IN2);
M033: NOP   0;
NETWORK
TITLE =

      A(    ;
      A(    ;
      A(    ;
      L     DIW   16;
      T     DIW 1122;
      SET   ;
      SAVE  ;
      CLR   ;
      A     BR;
      )     ;
      JNB   M034;
      L     DIW   18;
      T     DIW 1120;
      SET   ;
      SAVE  ;
      CLR   ;
M034: A     BR;
      )     ;
      JNB   M035;
      L     DIB   20;
      T     DIB 1125;
      SET   ;
      SAVE  ;
      CLR   ;
M035: A     BR;
      )     ;
      JNB   M036;
      L     DIB   21;
      T     DIB 1124;
M036: NOP   0;
NETWORK
TITLE =

      A(    ;
      A(    ;
      A(    ;
      L     DIB   22;
      T     DIB 1127;
      SET   ;
      SAVE  ;
      CLR   ;
      A     BR;
      )     ;
      JNB   M037;
      L     DIB   23;
      T     DIB 1126;
      SET   ;
      SAVE  ;
      CLR   ;
M037: A     BR;
      )     ;
      JNB   M038;
      L     DIB   24;
      T     DIB 1129;
      SET   ;
      SAVE  ;
      CLR   ;
M038: A     BR;
      )     ;
      JNB   M039;
      L     DIB   25;
      T     DIB 1128;
M039: NOP   0;
NETWORK
TITLE =

      A(    ;
      A(    ;
      A(    ;
      L     DIB   26;
      T     DIB 1131;
      SET   ;
      SAVE  ;
      CLR   ;
      A     BR;
      )     ;
      JNB   M03a;
      L     DIB   27;
      T     DIB 1130;
      SET   ;
      SAVE  ;
      CLR   ;
M03a: A     BR;
      )     ;
      JNB   M03b;
      L     DIB   28;
      T     DIB 1133;
      SET   ;
      SAVE  ;
      CLR   ;
M03b: A     BR;
      )     ;
      JNB   M03c;
      L     DIB   29;
      T     DIB 1132;
M03c: NOP   0;
END_FUNCTION

FUNCTION FC 506 : VOID
TITLE =
VERSION : 0.1

BEGIN
NETWORK
TITLE =
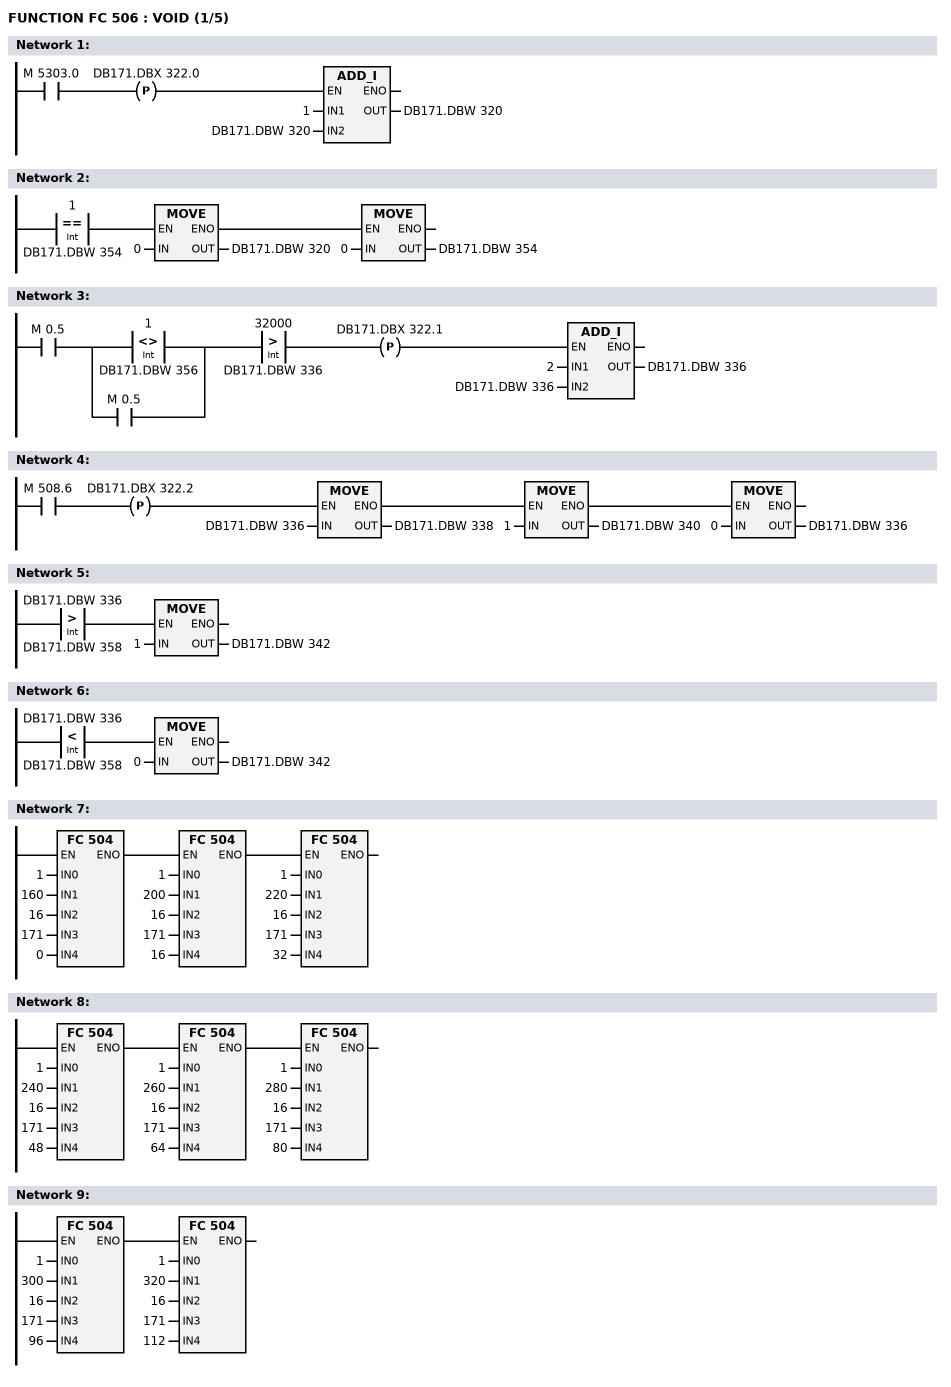

      A     M   5303.0;
      FP    DB171.DBX  322.0;
      JNB   _001;
      L     1;
      L     DB171.DBW  320;
      +I    ;
      T     DB171.DBW  320;
_001: NOP   0;
NETWORK
TITLE =

      A(    ;
      A(    ;
      L     1;
      L     DB171.DBW  354;
      ==I   ;
      )     ;
      JNB   _002;
      L     0;
      T     DB171.DBW  320;
      SET   ;
      SAVE  ;
      CLR   ;
_002: A     BR;
      )     ;
      JNB   _003;
      L     0;
      T     DB171.DBW  354;
_003: NOP   0;
NETWORK
TITLE =

      A     M      0.5;
      A(    ;
      O(    ;
      L     1;
      L     DB171.DBW  356;
      <>I   ;
      )     ;
      O     M      0.5;
      )     ;
      A(    ;
      L     32000;
      L     DB171.DBW  336;
      >I    ;
      )     ;
      FP    DB171.DBX  322.1;
      JNB   _004;
      L     2;
      L     DB171.DBW  336;
      +I    ;
      T     DB171.DBW  336;
_004: NOP   0;
NETWORK
TITLE =

      A(    ;
      A(    ;
      A     M    508.6;
      FP    DB171.DBX  322.2;
      JNB   _005;
      L     DB171.DBW  336;
      T     DB171.DBW  338;
      SET   ;
      SAVE  ;
      CLR   ;
_005: A     BR;
      )     ;
      JNB   _006;
      L     1;
      T     DB171.DBW  340;
      SET   ;
      SAVE  ;
      CLR   ;
_006: A     BR;
      )     ;
      JNB   _007;
      L     0;
      T     DB171.DBW  336;
_007: NOP   0;
NETWORK
TITLE =

      A(    ;
      L     DB171.DBW  336;
      L     DB171.DBW  358;
      >I    ;
      )     ;
      JNB   _008;
      L     1;
      T     DB171.DBW  342;
_008: NOP   0;
NETWORK
TITLE =

      A(    ;
      L     DB171.DBW  336;
      L     DB171.DBW  358;
      <I    ;
      )     ;
      JNB   _009;
      L     0;
      T     DB171.DBW  342;
_009: NOP   0;
NETWORK
TITLE =

      A(    ;
      A(    ;
      CALL FC   504 (
           IN0                      := 1,
           IN1                      := 160,
           IN2                      := 16,
           IN3                      := 171,
           IN4                      := 0);
      A     BR;
      )     ;
      JNB   _00a;
      CALL FC   504 (
           IN0                      := 1,
           IN1                      := 200,
           IN2                      := 16,
           IN3                      := 171,
           IN4                      := 16);
_00a: A     BR;
      )     ;
      JNB   _00b;
      CALL FC   504 (
           IN0                      := 1,
           IN1                      := 220,
           IN2                      := 16,
           IN3                      := 171,
           IN4                      := 32);
_00b: NOP   0;
NETWORK
TITLE =

      A(    ;
      A(    ;
      CALL FC   504 (
           IN0                      := 1,
           IN1                      := 240,
           IN2                      := 16,
           IN3                      := 171,
           IN4                      := 48);
      A     BR;
      )     ;
      JNB   _00c;
      CALL FC   504 (
           IN0                      := 1,
           IN1                      := 260,
           IN2                      := 16,
           IN3                      := 171,
           IN4                      := 64);
_00c: A     BR;
      )     ;
      JNB   _00d;
      CALL FC   504 (
           IN0                      := 1,
           IN1                      := 280,
           IN2                      := 16,
           IN3                      := 171,
           IN4                      := 80);
_00d: NOP   0;
NETWORK
TITLE =

      A(    ;
      CALL FC   504 (
           IN0                      := 1,
           IN1                      := 300,
           IN2                      := 16,
           IN3                      := 171,
           IN4                      := 96);
      A     BR;
      )     ;
      JNB   _00e;
      CALL FC   504 (
           IN0                      := 1,
           IN1                      := 320,
           IN2                      := 16,
           IN3                      := 171,
           IN4                      := 112);
_00e: NOP   0;
NETWORK
TITLE =
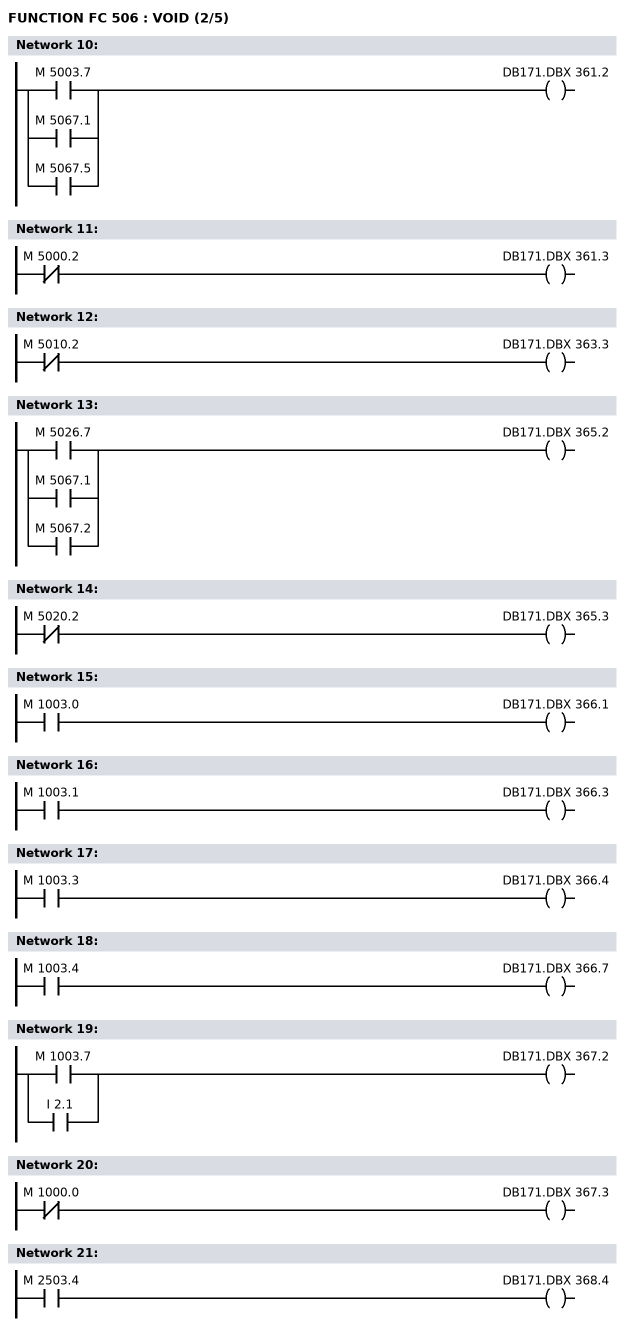

      O     M   5003.7;
      O     M   5067.1;
      O     M   5067.5;
      =     DB171.DBX  361.2;
NETWORK
TITLE =

      AN    M   5000.2;
      =     DB171.DBX  361.3;
NETWORK
TITLE =

      AN    M   5010.2;
      =     DB171.DBX  363.3;
NETWORK
TITLE =

      O     M   5026.7;
      O     M   5067.1;
      O     M   5067.2;
      =     DB171.DBX  365.2;
NETWORK
TITLE =

      AN    M   5020.2;
      =     DB171.DBX  365.3;
NETWORK
TITLE =

      A     M   1003.0;
      =     DB171.DBX  366.1;
NETWORK
TITLE =

      A     M   1003.1;
      =     DB171.DBX  366.3;
NETWORK
TITLE =

      A     M   1003.3;
      =     DB171.DBX  366.4;
NETWORK
TITLE =

      A     M   1003.4;
      =     DB171.DBX  366.7;
NETWORK
TITLE =

      O     M   1003.7;
      O     I      2.1;
      =     DB171.DBX  367.2;
NETWORK
TITLE =

      AN    M   1000.0;
      =     DB171.DBX  367.3;
NETWORK
TITLE =

      A     M   2503.4;
      =     DB171.DBX  368.4;
NETWORK
TITLE =
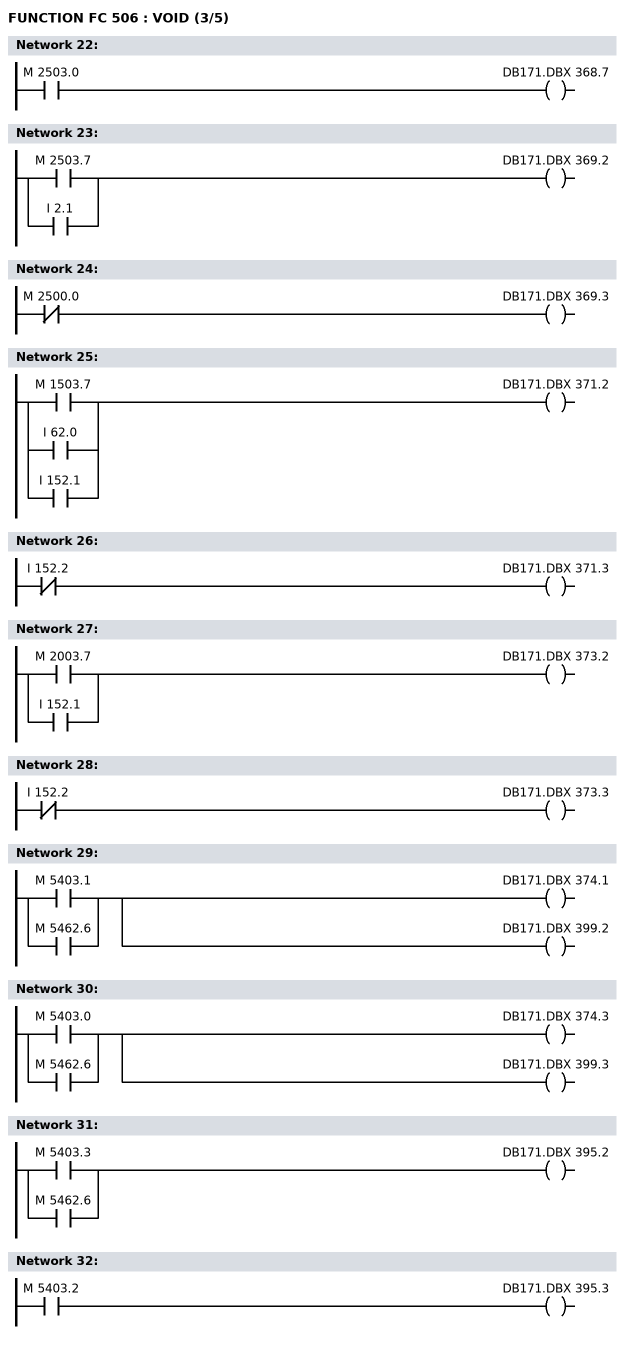

      A     M   2503.0;
      =     DB171.DBX  368.7;
NETWORK
TITLE =

      O     M   2503.7;
      O     I      2.1;
      =     DB171.DBX  369.2;
NETWORK
TITLE =

      AN    M   2500.0;
      =     DB171.DBX  369.3;
NETWORK
TITLE =

      O     M   1503.7;
      O     I     62.0;
      O     I    152.1;
      =     DB171.DBX  371.2;
NETWORK
TITLE =

      AN    I    152.2;
      =     DB171.DBX  371.3;
NETWORK
TITLE =

      O     M   2003.7;
      O     I    152.1;
      =     DB171.DBX  373.2;
NETWORK
TITLE =

      AN    I    152.2;
      =     DB171.DBX  373.3;
NETWORK
TITLE =

      O     M   5403.1;
      O     M   5462.6;
      =     DB171.DBX  374.1;
      =     DB171.DBX  399.2;
NETWORK
TITLE =

      O     M   5403.0;
      O     M   5462.6;
      =     DB171.DBX  374.3;
      =     DB171.DBX  399.3;
NETWORK
TITLE =

      O     M   5403.3;
      O     M   5462.6;
      =     DB171.DBX  395.2;
NETWORK
TITLE =

      A     M   5403.2;
      =     DB171.DBX  395.3;
NETWORK
TITLE =
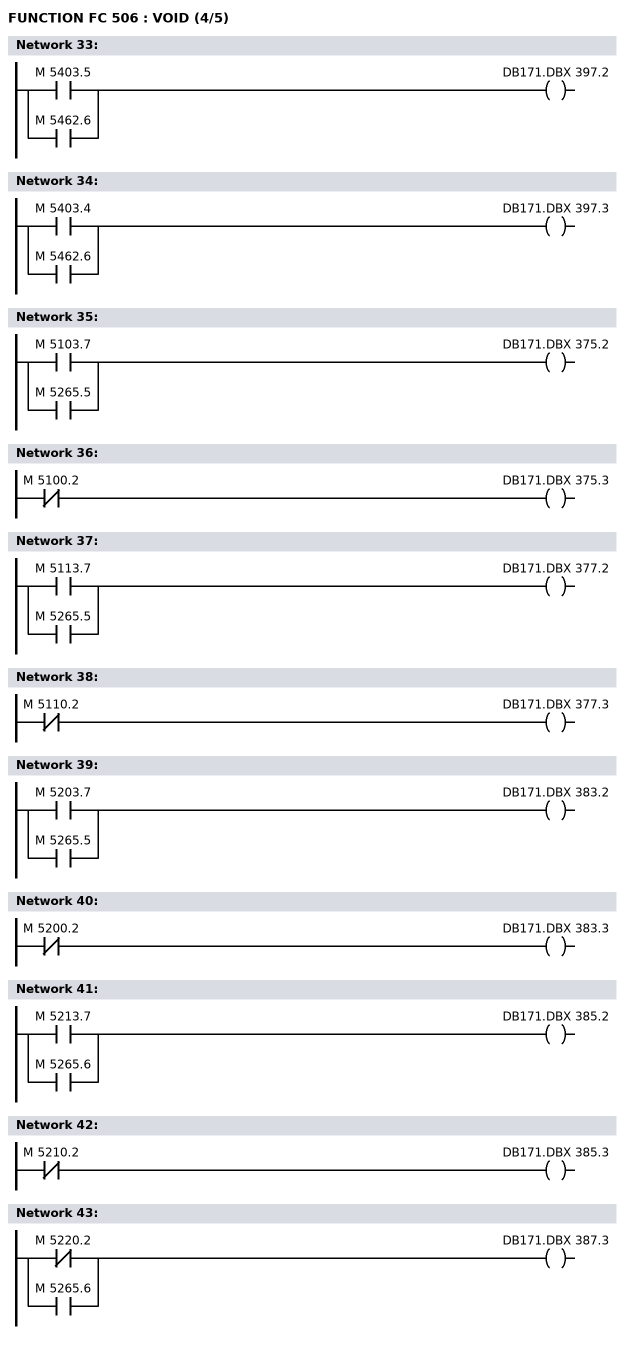

      O     M   5403.5;
      O     M   5462.6;
      =     DB171.DBX  397.2;
NETWORK
TITLE =

      O     M   5403.4;
      O     M   5462.6;
      =     DB171.DBX  397.3;
NETWORK
TITLE =

      O     M   5103.7;
      O     M   5265.5;
      =     DB171.DBX  375.2;
NETWORK
TITLE =

      AN    M   5100.2;
      =     DB171.DBX  375.3;
NETWORK
TITLE =

      O     M   5113.7;
      O     M   5265.5;
      =     DB171.DBX  377.2;
NETWORK
TITLE =

      AN    M   5110.2;
      =     DB171.DBX  377.3;
NETWORK
TITLE =

      O     M   5203.7;
      O     M   5265.5;
      =     DB171.DBX  383.2;
NETWORK
TITLE =

      AN    M   5200.2;
      =     DB171.DBX  383.3;
NETWORK
TITLE =

      O     M   5213.7;
      O     M   5265.6;
      =     DB171.DBX  385.2;
NETWORK
TITLE =

      AN    M   5210.2;
      =     DB171.DBX  385.3;
NETWORK
TITLE =

      ON    M   5220.2;
      O     M   5265.6;
      =     DB171.DBX  387.3;
NETWORK
TITLE =
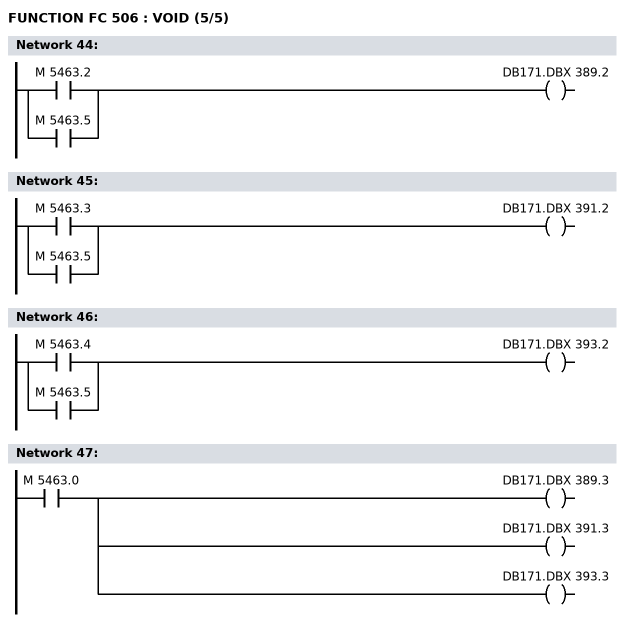

      O     M   5463.2;
      O     M   5463.5;
      =     DB171.DBX  389.2;
NETWORK
TITLE =

      O     M   5463.3;
      O     M   5463.5;
      =     DB171.DBX  391.2;
NETWORK
TITLE =

      O     M   5463.4;
      O     M   5463.5;
      =     DB171.DBX  393.2;
NETWORK
TITLE =

      A     M   5463.0;
      =     DB171.DBX  389.3;
      =     DB171.DBX  391.3;
      =     DB171.DBX  393.3;
NETWORK
TITLE =

      AN    OV;
      A(    ;
      O     M    304.0;
      O     M    304.1;
      )     ;
      A     M   1002.0;
      FP    M     20.1;
      JNB   _00f;
      L     1;
      T     DB171.DBW  202;
_00f: NOP   0;
NETWORK
TITLE =
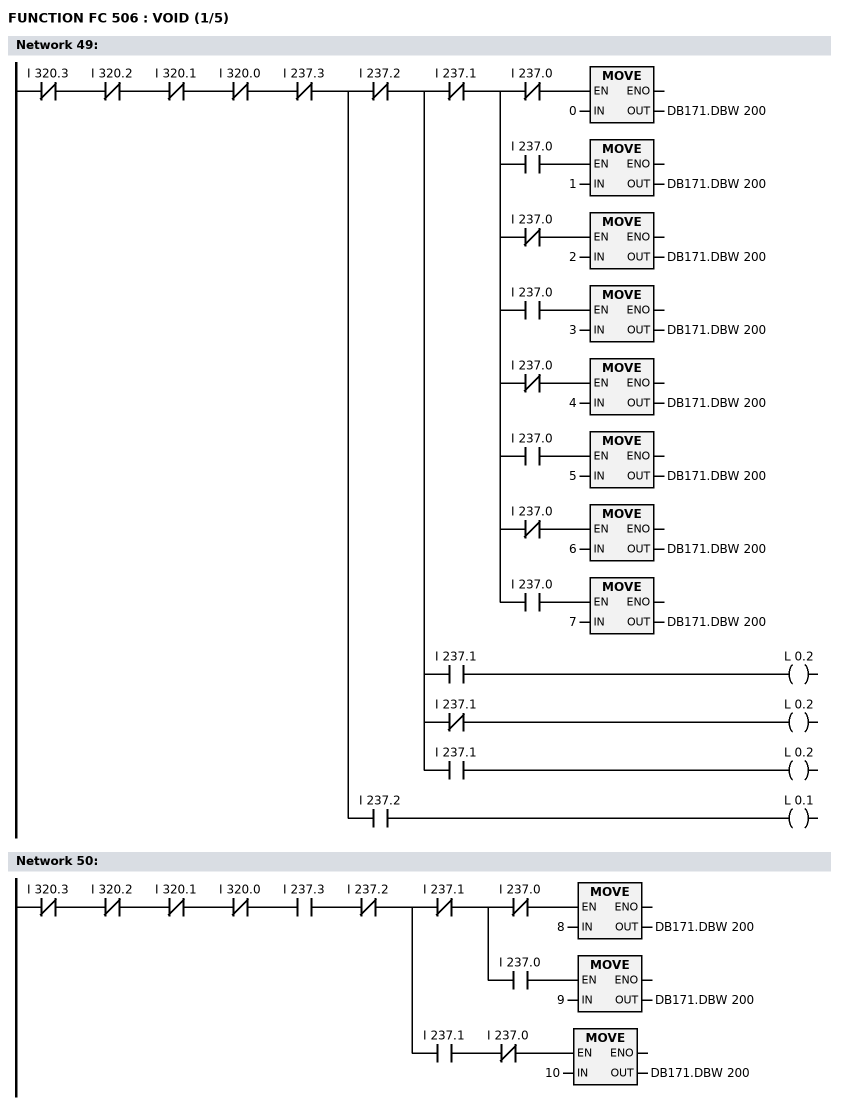

      AN    I    320.3;
      AN    I    320.2;
      AN    I    320.1;
      AN    I    320.0;
      AN    I    237.3;
      =     L      0.0;
      A     L      0.0;
      AN    I    237.2;
      =     L      0.1;
      A     L      0.1;
      AN    I    237.1;
      =     L      0.2;
      A     L      0.2;
      AN    I    237.0;
      JNB   _010;
      L     0;
      T     DB171.DBW  200;
_010: NOP   0;
      A     L      0.2;
      A     I    237.0;
      JNB   _011;
      L     1;
      T     DB171.DBW  200;
_011: NOP   0;
      A     L      0.1;
      A     I    237.1;
      =     L      0.2;
      A     L      0.2;
      AN    I    237.0;
      JNB   _012;
      L     2;
      T     DB171.DBW  200;
_012: NOP   0;
      A     L      0.2;
      A     I    237.0;
      JNB   _013;
      L     3;
      T     DB171.DBW  200;
_013: NOP   0;
      A     L      0.0;
      A     I    237.2;
      =     L      0.1;
      A     L      0.1;
      AN    I    237.1;
      =     L      0.2;
      A     L      0.2;
      AN    I    237.0;
      JNB   _014;
      L     4;
      T     DB171.DBW  200;
_014: NOP   0;
      A     L      0.2;
      A     I    237.0;
      JNB   _015;
      L     5;
      T     DB171.DBW  200;
_015: NOP   0;
      A     L      0.1;
      A     I    237.1;
      =     L      0.2;
      A     L      0.2;
      AN    I    237.0;
      JNB   _016;
      L     6;
      T     DB171.DBW  200;
_016: NOP   0;
      A     L      0.2;
      A     I    237.0;
      JNB   _017;
      L     7;
      T     DB171.DBW  200;
_017: NOP   0;
NETWORK
TITLE =

      AN    I    320.3;
      AN    I    320.2;
      AN    I    320.1;
      AN    I    320.0;
      A     I    237.3;
      AN    I    237.2;
      =     L      0.0;
      A     L      0.0;
      AN    I    237.1;
      =     L      0.1;
      A     L      0.1;
      AN    I    237.0;
      JNB   _018;
      L     8;
      T     DB171.DBW  200;
_018: NOP   0;
      A     L      0.1;
      A     I    237.0;
      JNB   _019;
      L     9;
      T     DB171.DBW  200;
_019: NOP   0;
      A     L      0.0;
      A     I    237.1;
      AN    I    237.0;
      JNB   _01a;
      L     10;
      T     DB171.DBW  200;
_01a: NOP   0;
NETWORK
TITLE =
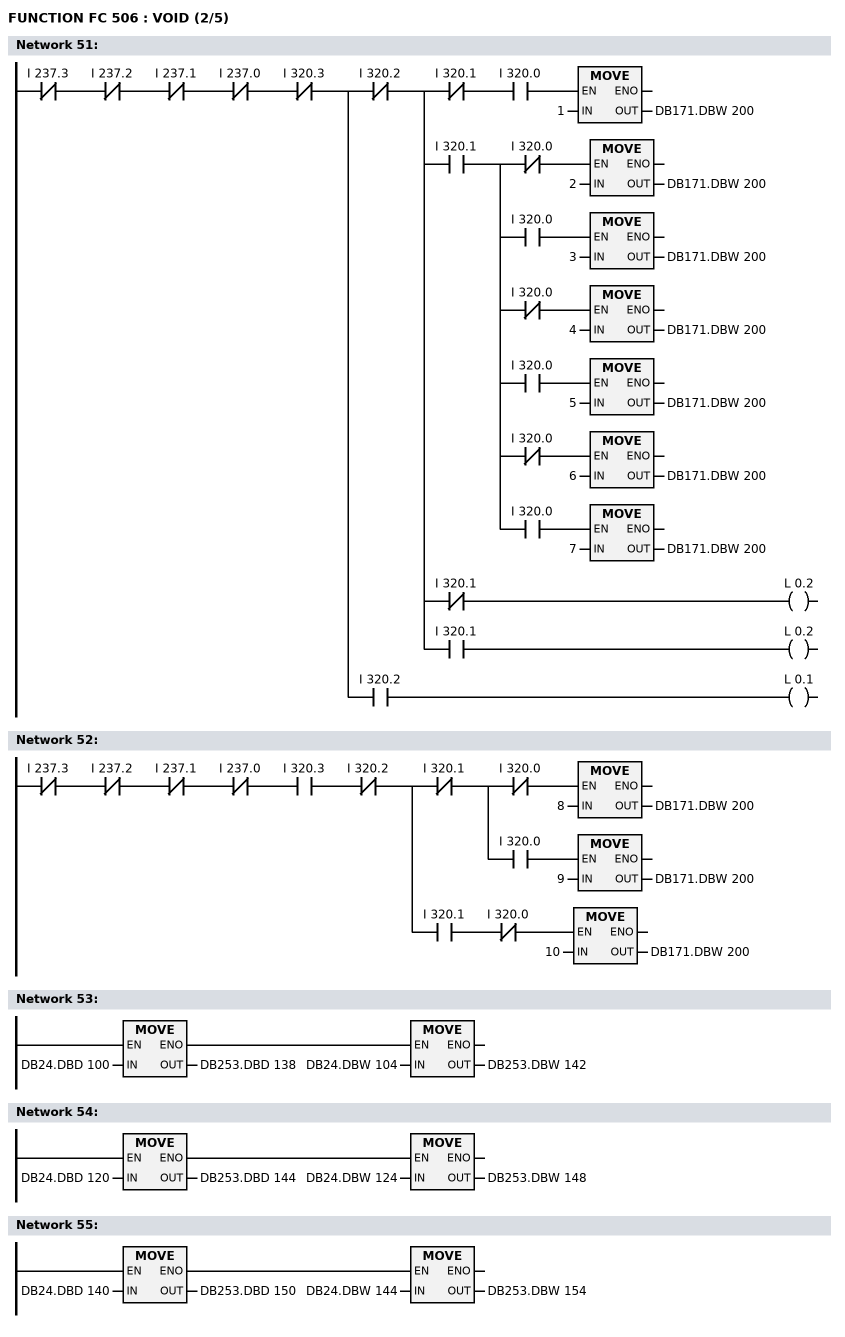

      AN    I    237.3;
      AN    I    237.2;
      AN    I    237.1;
      AN    I    237.0;
      AN    I    320.3;
      =     L      0.0;
      A     L      0.0;
      AN    I    320.2;
      =     L      0.1;
      A     L      0.1;
      AN    I    320.1;
      A     I    320.0;
      JNB   _01b;
      L     1;
      T     DB171.DBW  200;
_01b: NOP   0;
      A     L      0.1;
      A     I    320.1;
      =     L      0.2;
      A     L      0.2;
      AN    I    320.0;
      JNB   _01c;
      L     2;
      T     DB171.DBW  200;
_01c: NOP   0;
      A     L      0.2;
      A     I    320.0;
      JNB   _01d;
      L     3;
      T     DB171.DBW  200;
_01d: NOP   0;
      A     L      0.0;
      A     I    320.2;
      =     L      0.1;
      A     L      0.1;
      AN    I    320.1;
      =     L      0.2;
      A     L      0.2;
      AN    I    320.0;
      JNB   _01e;
      L     4;
      T     DB171.DBW  200;
_01e: NOP   0;
      A     L      0.2;
      A     I    320.0;
      JNB   _01f;
      L     5;
      T     DB171.DBW  200;
_01f: NOP   0;
      A     L      0.1;
      A     I    320.1;
      =     L      0.2;
      A     L      0.2;
      AN    I    320.0;
      JNB   _020;
      L     6;
      T     DB171.DBW  200;
_020: NOP   0;
      A     L      0.2;
      A     I    320.0;
      JNB   _021;
      L     7;
      T     DB171.DBW  200;
_021: NOP   0;
NETWORK
TITLE =

      AN    I    237.3;
      AN    I    237.2;
      AN    I    237.1;
      AN    I    237.0;
      A     I    320.3;
      AN    I    320.2;
      =     L      0.0;
      A     L      0.0;
      AN    I    320.1;
      =     L      0.1;
      A     L      0.1;
      AN    I    320.0;
      JNB   _022;
      L     8;
      T     DB171.DBW  200;
_022: NOP   0;
      A     L      0.1;
      A     I    320.0;
      JNB   _023;
      L     9;
      T     DB171.DBW  200;
_023: NOP   0;
      A     L      0.0;
      A     I    320.1;
      AN    I    320.0;
      JNB   _024;
      L     10;
      T     DB171.DBW  200;
_024: NOP   0;
NETWORK
TITLE =

      A(    ;
      L     DB24.DBD  100;
      T     DB253.DBD  138;
      SET   ;
      SAVE  ;
      CLR   ;
      A     BR;
      )     ;
      JNB   _025;
      L     DB24.DBW  104;
      T     DB253.DBW  142;
_025: NOP   0;
NETWORK
TITLE =

      A(    ;
      L     DB24.DBD  120;
      T     DB253.DBD  144;
      SET   ;
      SAVE  ;
      CLR   ;
      A     BR;
      )     ;
      JNB   _026;
      L     DB24.DBW  124;
      T     DB253.DBW  148;
_026: NOP   0;
NETWORK
TITLE =

      A(    ;
      L     DB24.DBD  140;
      T     DB253.DBD  150;
      SET   ;
      SAVE  ;
      CLR   ;
      A     BR;
      )     ;
      JNB   _027;
      L     DB24.DBW  144;
      T     DB253.DBW  154;
_027: NOP   0;
NETWORK
TITLE =
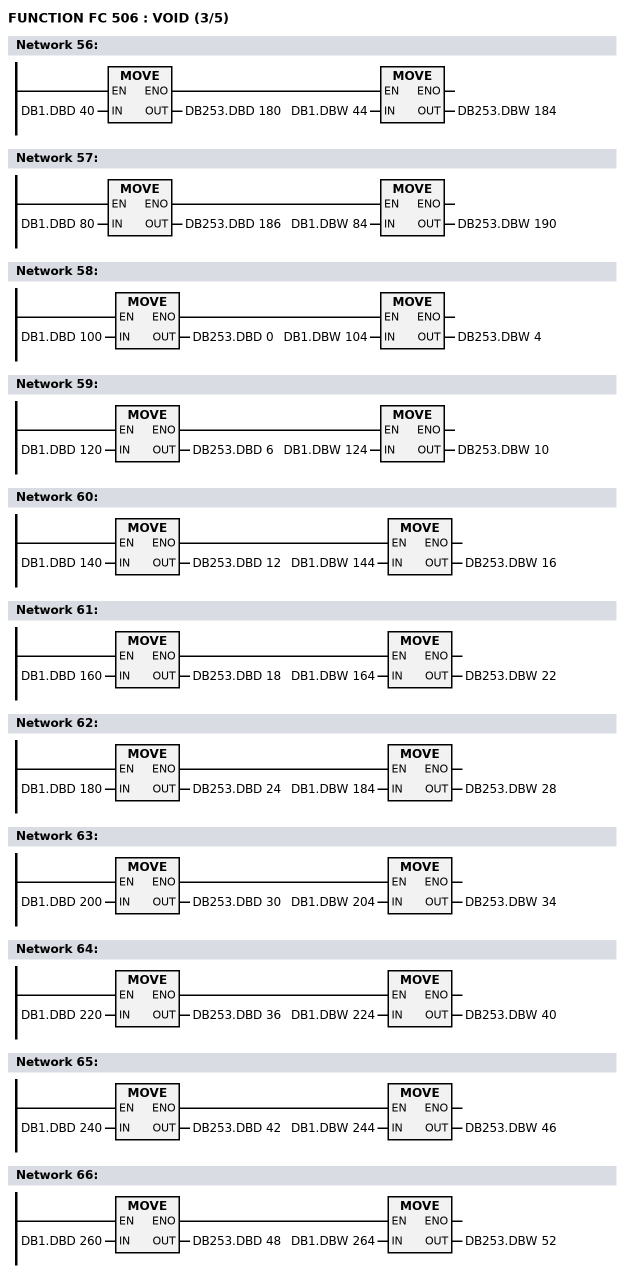

      A(    ;
      L     DB1.DBD   40;
      T     DB253.DBD  180;
      SET   ;
      SAVE  ;
      CLR   ;
      A     BR;
      )     ;
      JNB   _028;
      L     DB1.DBW   44;
      T     DB253.DBW  184;
_028: NOP   0;
NETWORK
TITLE =

      A(    ;
      L     DB1.DBD   80;
      T     DB253.DBD  186;
      SET   ;
      SAVE  ;
      CLR   ;
      A     BR;
      )     ;
      JNB   _029;
      L     DB1.DBW   84;
      T     DB253.DBW  190;
_029: NOP   0;
NETWORK
TITLE =

      A(    ;
      L     DB1.DBD  100;
      T     DB253.DBD    0;
      SET   ;
      SAVE  ;
      CLR   ;
      A     BR;
      )     ;
      JNB   _02a;
      L     DB1.DBW  104;
      T     DB253.DBW    4;
_02a: NOP   0;
NETWORK
TITLE =

      A(    ;
      L     DB1.DBD  120;
      T     DB253.DBD    6;
      SET   ;
      SAVE  ;
      CLR   ;
      A     BR;
      )     ;
      JNB   _02b;
      L     DB1.DBW  124;
      T     DB253.DBW   10;
_02b: NOP   0;
NETWORK
TITLE =

      A(    ;
      L     DB1.DBD  140;
      T     DB253.DBD   12;
      SET   ;
      SAVE  ;
      CLR   ;
      A     BR;
      )     ;
      JNB   _02c;
      L     DB1.DBW  144;
      T     DB253.DBW   16;
_02c: NOP   0;
NETWORK
TITLE =

      A(    ;
      L     DB1.DBD  160;
      T     DB253.DBD   18;
      SET   ;
      SAVE  ;
      CLR   ;
      A     BR;
      )     ;
      JNB   _02d;
      L     DB1.DBW  164;
      T     DB253.DBW   22;
_02d: NOP   0;
NETWORK
TITLE =

      A(    ;
      L     DB1.DBD  180;
      T     DB253.DBD   24;
      SET   ;
      SAVE  ;
      CLR   ;
      A     BR;
      )     ;
      JNB   _02e;
      L     DB1.DBW  184;
      T     DB253.DBW   28;
_02e: NOP   0;
NETWORK
TITLE =

      A(    ;
      L     DB1.DBD  200;
      T     DB253.DBD   30;
      SET   ;
      SAVE  ;
      CLR   ;
      A     BR;
      )     ;
      JNB   _02f;
      L     DB1.DBW  204;
      T     DB253.DBW   34;
_02f: NOP   0;
NETWORK
TITLE =

      A(    ;
      L     DB1.DBD  220;
      T     DB253.DBD   36;
      SET   ;
      SAVE  ;
      CLR   ;
      A     BR;
      )     ;
      JNB   _030;
      L     DB1.DBW  224;
      T     DB253.DBW   40;
_030: NOP   0;
NETWORK
TITLE =

      A(    ;
      L     DB1.DBD  240;
      T     DB253.DBD   42;
      SET   ;
      SAVE  ;
      CLR   ;
      A     BR;
      )     ;
      JNB   _031;
      L     DB1.DBW  244;
      T     DB253.DBW   46;
_031: NOP   0;
NETWORK
TITLE =

      A(    ;
      L     DB1.DBD  260;
      T     DB253.DBD   48;
      SET   ;
      SAVE  ;
      CLR   ;
      A     BR;
      )     ;
      JNB   _032;
      L     DB1.DBW  264;
      T     DB253.DBW   52;
_032: NOP   0;
NETWORK
TITLE =
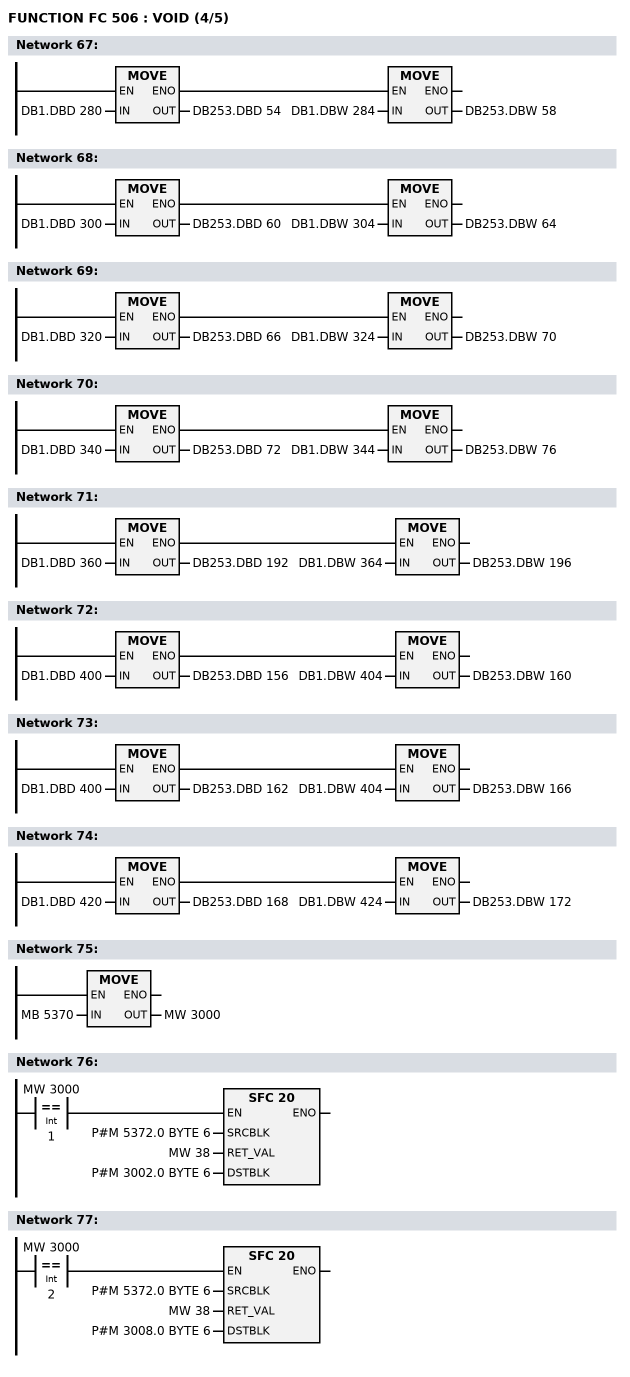

      A(    ;
      L     DB1.DBD  280;
      T     DB253.DBD   54;
      SET   ;
      SAVE  ;
      CLR   ;
      A     BR;
      )     ;
      JNB   _033;
      L     DB1.DBW  284;
      T     DB253.DBW   58;
_033: NOP   0;
NETWORK
TITLE =

      A(    ;
      L     DB1.DBD  300;
      T     DB253.DBD   60;
      SET   ;
      SAVE  ;
      CLR   ;
      A     BR;
      )     ;
      JNB   _034;
      L     DB1.DBW  304;
      T     DB253.DBW   64;
_034: NOP   0;
NETWORK
TITLE =

      A(    ;
      L     DB1.DBD  320;
      T     DB253.DBD   66;
      SET   ;
      SAVE  ;
      CLR   ;
      A     BR;
      )     ;
      JNB   _035;
      L     DB1.DBW  324;
      T     DB253.DBW   70;
_035: NOP   0;
NETWORK
TITLE =

      A(    ;
      L     DB1.DBD  340;
      T     DB253.DBD   72;
      SET   ;
      SAVE  ;
      CLR   ;
      A     BR;
      )     ;
      JNB   _036;
      L     DB1.DBW  344;
      T     DB253.DBW   76;
_036: NOP   0;
NETWORK
TITLE =

      A(    ;
      L     DB1.DBD  360;
      T     DB253.DBD  192;
      SET   ;
      SAVE  ;
      CLR   ;
      A     BR;
      )     ;
      JNB   _037;
      L     DB1.DBW  364;
      T     DB253.DBW  196;
_037: NOP   0;
NETWORK
TITLE =

      A(    ;
      L     DB1.DBD  400;
      T     DB253.DBD  156;
      SET   ;
      SAVE  ;
      CLR   ;
      A     BR;
      )     ;
      JNB   _038;
      L     DB1.DBW  404;
      T     DB253.DBW  160;
_038: NOP   0;
NETWORK
TITLE =

      A(    ;
      L     DB1.DBD  400;
      T     DB253.DBD  162;
      SET   ;
      SAVE  ;
      CLR   ;
      A     BR;
      )     ;
      JNB   _039;
      L     DB1.DBW  404;
      T     DB253.DBW  166;
_039: NOP   0;
NETWORK
TITLE =

      A(    ;
      L     DB1.DBD  420;
      T     DB253.DBD  168;
      SET   ;
      SAVE  ;
      CLR   ;
      A     BR;
      )     ;
      JNB   _03a;
      L     DB1.DBW  424;
      T     DB253.DBW  172;
_03a: NOP   0;
NETWORK
TITLE =

      L     MB  5370;
      T     MW  3000;
      NOP   0;
NETWORK
TITLE =

      A(    ;
      L     MW  3000;
      L     1;
      ==I   ;
      )     ;
      JNB   _03b;
      CALL SFC   20 (
           SRCBLK                   := P#M 5372.0 BYTE 6,
           RET_VAL                  := MW    38,
           DSTBLK                   := P#M 3002.0 BYTE 6);
_03b: NOP   0;
NETWORK
TITLE =

      A(    ;
      L     MW  3000;
      L     2;
      ==I   ;
      )     ;
      JNB   _03c;
      CALL SFC   20 (
           SRCBLK                   := P#M 5372.0 BYTE 6,
           RET_VAL                  := MW    38,
           DSTBLK                   := P#M 3008.0 BYTE 6);
_03c: NOP   0;
NETWORK
TITLE =
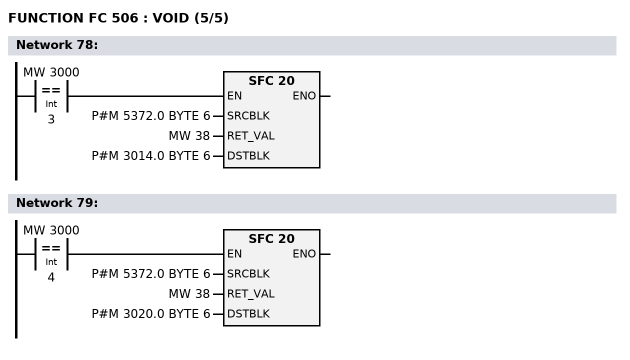

      A(    ;
      L     MW  3000;
      L     3;
      ==I   ;
      )     ;
      JNB   _03d;
      CALL SFC   20 (
           SRCBLK                   := P#M 5372.0 BYTE 6,
           RET_VAL                  := MW    38,
           DSTBLK                   := P#M 3014.0 BYTE 6);
_03d: NOP   0;
NETWORK
TITLE =

      A(    ;
      L     MW  3000;
      L     4;
      ==I   ;
      )     ;
      JNB   _03e;
      CALL SFC   20 (
           SRCBLK                   := P#M 5372.0 BYTE 6,
           RET_VAL                  := MW    38,
           DSTBLK                   := P#M 3020.0 BYTE 6);
_03e: NOP   0;
NETWORK
TITLE =

      AN    OV;
      JNB   _03f;
      CALL SFC   20 (
           SRCBLK                   := P#M 3002.0 BYTE 24,
           RET_VAL                  := MW    38,
           DSTBLK                   := P#DB253.DBX78.0 BYTE 24);
_03f: NOP   0;
END_FUNCTION

FUNCTION FC 510 : VOID
TITLE =
VERSION : 0.1


VAR_INPUT
  IN0 : INT ;
  IN1 : INT ;
  IN2 : INT ;
  IN3 : INT ;
  IN4 : INT ;
  IN5 : INT ;
  IN6 : INT ;
  IN7 : BOOL ;
  IN8 : BOOL ;
  IN9 : BOOL ;
  IN10 : BOOL ;
  IN11 : BOOL ;
  IN12 : BOOL ;
END_VAR
VAR_OUTPUT
  OUT13 : BOOL ;
  OUT14 : BOOL ;
END_VAR
VAR_TEMP
  TEMP15 : INT ;
  TEMP16 : INT ;
  TEMP17 : INT ;
  TEMP18 : INT ;
  TEMP19 : INT ;
  TEMP20 : INT ;
  TEMP21 : INT ;
  TEMP22 : BOOL ;
  TEMP23 : WORD ;
  TEMP24 : WORD ;
  TEMP25 : INT ;
  TEMP26 : WORD ;
  TEMP27 : INT ;
  TEMP28 : INT ;
  TEMP29 : INT ;
  TEMP30 : INT ;
END_VAR
BEGIN
NETWORK
TITLE =

      L     #IN0;
      T     #TEMP15;
      L     #IN1;
      T     #TEMP16;
      L     #IN2;
      T     #TEMP17;
      L     #IN3;
      T     #TEMP18;
      OPN   DI [#TEMP17];
NETWORK
TITLE =

      CALL FC   504 (
           IN0                      := #TEMP18,
           IN1                      := #IN4,
           IN2                      := 16,
           IN3                      := #TEMP17,
           IN4                      := 16);
      NOP   0;
NETWORK
TITLE =

      A(    ;
      L     DIW   17;
      L     DIW   18;
      OW    ;
      T     #TEMP24;
      SET   ;
      SAVE  ;
      CLR   ;
      A     BR;
      )     ;
      JNB   _001;
      L     DIW   18;
      T     #TEMP24;
_001: NOP   0;
NETWORK
TITLE =

      A(    ;
      L     60;
      L     #TEMP15;
      *I    ;
      T     #TEMP20;
      AN    OV;
      SAVE  ;
      CLR   ;
      A     BR;
      )     ;
      JNB   _002;
      L     #TEMP20;
      L     60;
      -I    ;
      T     #TEMP21;
_002: NOP   0;
NETWORK
TITLE =

      O(    ;
      L     0;
      L     #TEMP15;
      ==I   ;
      )     ;
      O(    ;
      L     16;
      L     #TEMP15;
      <I    ;
      )     ;
      SAVE  ;
      BEC   ;
NETWORK
TITLE =

      OPN   DB [#TEMP16];
      L     #TEMP21;
      SLW   3;
      LAR1  ;
NETWORK
TITLE =
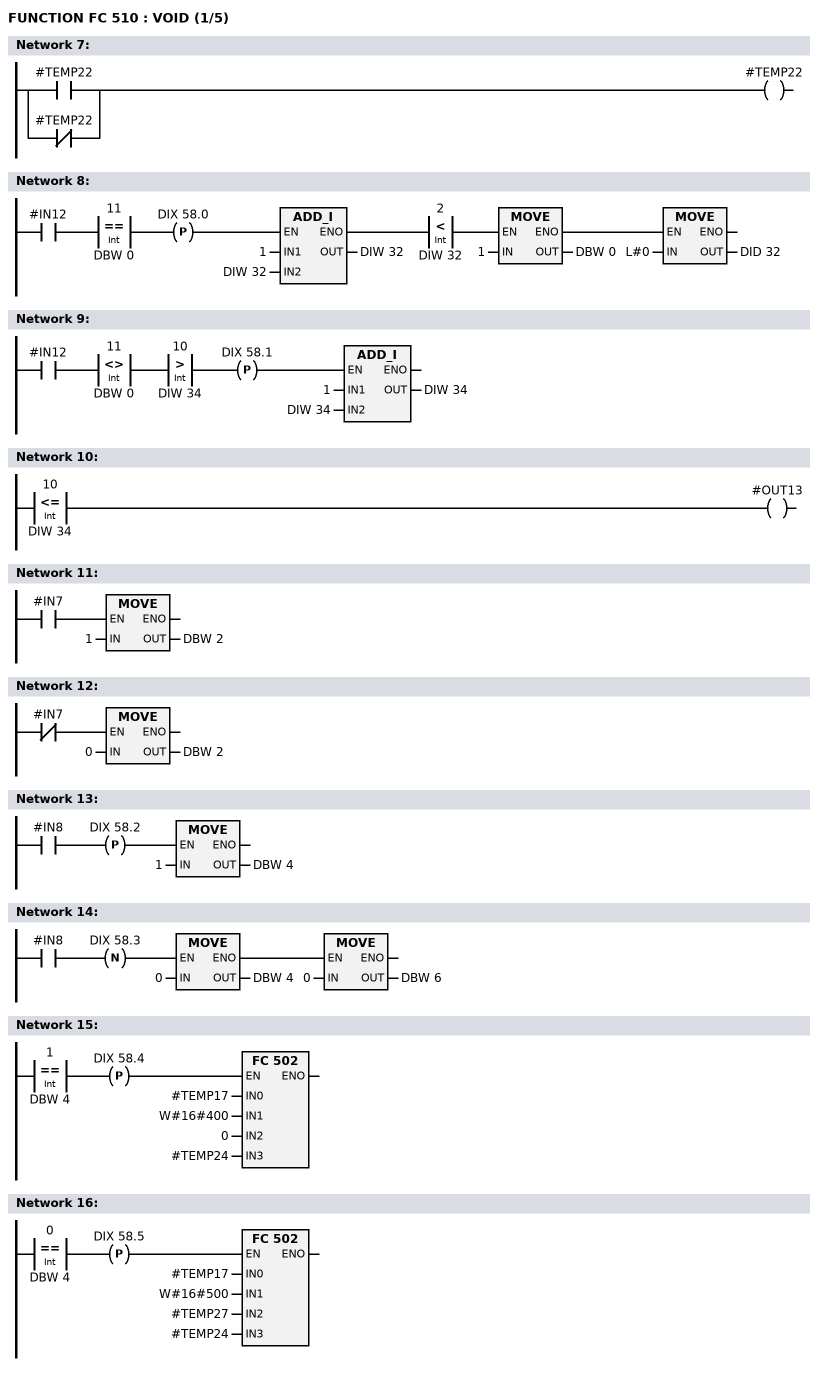

      O     #TEMP22;
      ON    #TEMP22;
      =     #TEMP22;
NETWORK
TITLE =

      A(    ;
      A(    ;
      A     #IN12;
      A(    ;
      L     11;
      L     DBW    0;
      ==I   ;
      )     ;
      FP    DIX   58.0;
      JNB   _003;
      L     1;
      L     DIW   32;
      +I    ;
      T     DIW   32;
      AN    OV;
      SAVE  ;
      CLR   ;
_003: A     BR;
      )     ;
      A(    ;
      L     2;
      L     DIW   32;
      <I    ;
      )     ;
      JNB   _004;
      L     1;
      T     DBW    0;
      SET   ;
      SAVE  ;
      CLR   ;
_004: A     BR;
      )     ;
      JNB   _005;
      L     L#0;
      T     DID   32;
_005: NOP   0;
NETWORK
TITLE =

      A     #IN12;
      A(    ;
      L     11;
      L     DBW    0;
      <>I   ;
      )     ;
      A(    ;
      L     10;
      L     DIW   34;
      >I    ;
      )     ;
      FP    DIX   58.1;
      JNB   _006;
      L     1;
      L     DIW   34;
      +I    ;
      T     DIW   34;
_006: NOP   0;
NETWORK
TITLE =

      L     10;
      L     DIW   34;
      <=I   ;
      =     #OUT13;
NETWORK
TITLE =

      A     #IN7;
      JNB   _007;
      L     1;
      T     DBW    2;
_007: NOP   0;
NETWORK
TITLE =

      AN    #IN7;
      JNB   _008;
      L     0;
      T     DBW    2;
_008: NOP   0;
NETWORK
TITLE =

      A     #IN8;
      FP    DIX   58.2;
      JNB   _009;
      L     1;
      T     DBW    4;
_009: NOP   0;
NETWORK
TITLE =

      A(    ;
      A     #IN8;
      FN    DIX   58.3;
      JNB   _00a;
      L     0;
      T     DBW    4;
      SET   ;
      SAVE  ;
      CLR   ;
_00a: A     BR;
      )     ;
      JNB   _00b;
      L     0;
      T     DBW    6;
_00b: NOP   0;
NETWORK
TITLE =

      A(    ;
      L     1;
      L     DBW    4;
      ==I   ;
      )     ;
      FP    DIX   58.4;
      JNB   _00c;
      CALL FC   502 (
           IN0                      := #TEMP17,
           IN1                      := W#16#400,
           IN2                      := 0,
           IN3                      := #TEMP24);
_00c: NOP   0;
NETWORK
TITLE =

      A(    ;
      L     0;
      L     DBW    4;
      ==I   ;
      )     ;
      FP    DIX   58.5;
      JNB   _00d;
      CALL FC   502 (
           IN0                      := #TEMP17,
           IN1                      := W#16#500,
           IN2                      := #TEMP27,
           IN3                      := #TEMP24);
_00d: NOP   0;
NETWORK
TITLE =
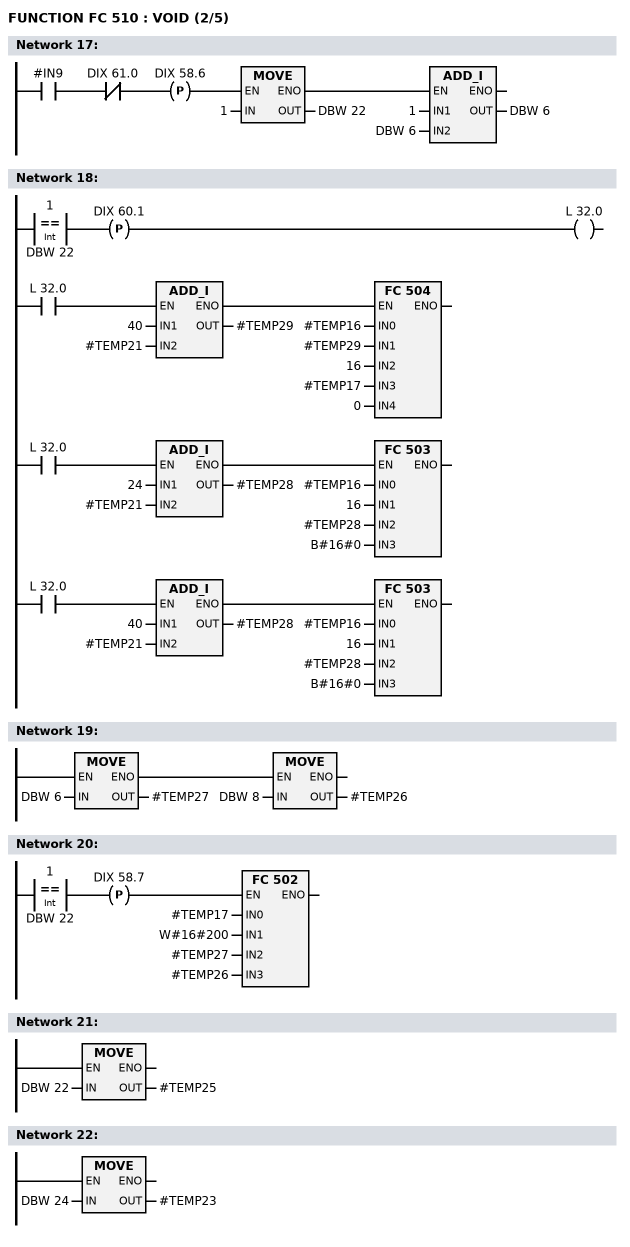

      A(    ;
      A     #IN9;
      AN    DIX   61.0;
      FP    DIX   58.6;
      JNB   _00e;
      L     1;
      T     DBW   22;
      SET   ;
      SAVE  ;
      CLR   ;
_00e: A     BR;
      )     ;
      JNB   _00f;
      L     1;
      L     DBW    6;
      +I    ;
      T     DBW    6;
_00f: NOP   0;
NETWORK
TITLE =

      A(    ;
      L     1;
      L     DBW   22;
      ==I   ;
      )     ;
      FP    DIX   60.1;
      =     L     32.0;
      A(    ;
      A     L     32.0;
      JNB   _010;
      L     40;
      L     #TEMP21;
      +I    ;
      T     #TEMP29;
      AN    OV;
      SAVE  ;
      CLR   ;
_010: A     BR;
      )     ;
      JNB   _011;
      CALL FC   504 (
           IN0                      := #TEMP16,
           IN1                      := #TEMP29,
           IN2                      := 16,
           IN3                      := #TEMP17,
           IN4                      := 0);
_011: NOP   0;
      A(    ;
      A     L     32.0;
      JNB   _012;
      L     24;
      L     #TEMP21;
      +I    ;
      T     #TEMP28;
      AN    OV;
      SAVE  ;
      CLR   ;
_012: A     BR;
      )     ;
      JNB   _013;
      CALL FC   503 (
           IN0                      := #TEMP16,
           IN1                      := 16,
           IN2                      := #TEMP28,
           IN3                      := B#16#0);
_013: NOP   0;
      A(    ;
      A     L     32.0;
      JNB   _014;
      L     40;
      L     #TEMP21;
      +I    ;
      T     #TEMP28;
      AN    OV;
      SAVE  ;
      CLR   ;
_014: A     BR;
      )     ;
      JNB   _015;
      CALL FC   503 (
           IN0                      := #TEMP16,
           IN1                      := 16,
           IN2                      := #TEMP28,
           IN3                      := B#16#0);
_015: NOP   0;
NETWORK
TITLE =

      A(    ;
      L     DBW    6;
      T     #TEMP27;
      SET   ;
      SAVE  ;
      CLR   ;
      A     BR;
      )     ;
      JNB   _016;
      L     DBW    8;
      T     #TEMP26;
_016: NOP   0;
NETWORK
TITLE =

      A(    ;
      L     1;
      L     DBW   22;
      ==I   ;
      )     ;
      FP    DIX   58.7;
      JNB   _017;
      CALL FC   502 (
           IN0                      := #TEMP17,
           IN1                      := W#16#200,
           IN2                      := #TEMP27,
           IN3                      := #TEMP26);
_017: NOP   0;
NETWORK
TITLE =

      L     DBW   22;
      T     #TEMP25;
      NOP   0;
NETWORK
TITLE =

      L     DBW   24;
      T     #TEMP23;
      NOP   0;
NETWORK
TITLE =
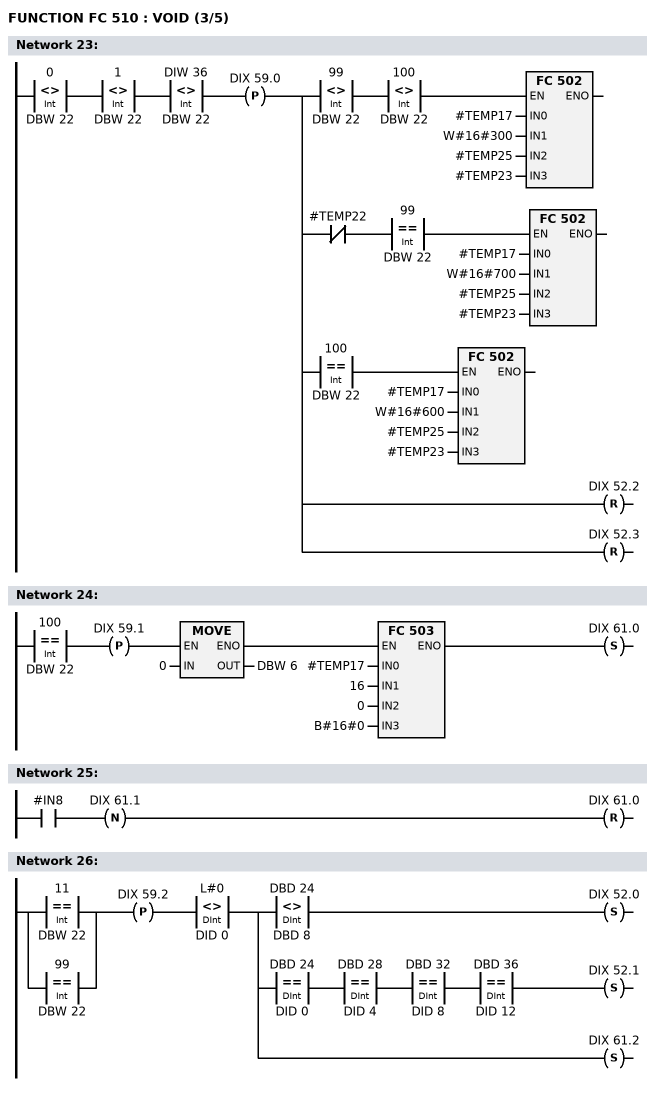

      A(    ;
      L     0;
      L     DBW   22;
      <>I   ;
      )     ;
      A(    ;
      L     1;
      L     DBW   22;
      <>I   ;
      )     ;
      A(    ;
      L     DIW   36;
      L     DBW   22;
      <>I   ;
      )     ;
      FP    DIX   59.0;
      =     L     32.0;
      A     L     32.0;
      A(    ;
      L     99;
      L     DBW   22;
      <>I   ;
      )     ;
      A(    ;
      L     100;
      L     DBW   22;
      <>I   ;
      )     ;
      JNB   _018;
      CALL FC   502 (
           IN0                      := #TEMP17,
           IN1                      := W#16#300,
           IN2                      := #TEMP25,
           IN3                      := #TEMP23);
_018: NOP   0;
      A     L     32.0;
      AN    #TEMP22;
      A(    ;
      L     99;
      L     DBW   22;
      ==I   ;
      )     ;
      JNB   _019;
      CALL FC   502 (
           IN0                      := #TEMP17,
           IN1                      := W#16#700,
           IN2                      := #TEMP25,
           IN3                      := #TEMP23);
_019: NOP   0;
      A     L     32.0;
      A(    ;
      L     100;
      L     DBW   22;
      ==I   ;
      )     ;
      JNB   _01a;
      CALL FC   502 (
           IN0                      := #TEMP17,
           IN1                      := W#16#600,
           IN2                      := #TEMP25,
           IN3                      := #TEMP23);
_01a: NOP   0;
      A     L     32.0;
      BLD   102;
      R     DIX   52.2;
      A     L     32.0;
      BLD   102;
      R     DIX   52.3;
NETWORK
TITLE =

      A(    ;
      A(    ;
      L     100;
      L     DBW   22;
      ==I   ;
      )     ;
      FP    DIX   59.1;
      JNB   _01b;
      L     0;
      T     DBW    6;
      SET   ;
      SAVE  ;
      CLR   ;
_01b: A     BR;
      )     ;
      JNB   _01c;
      CALL FC   503 (
           IN0                      := #TEMP17,
           IN1                      := 16,
           IN2                      := 0,
           IN3                      := B#16#0);
_01c: A     BR;
      S     DIX   61.0;
NETWORK
TITLE =

      A     #IN8;
      FN    DIX   61.1;
      R     DIX   61.0;
NETWORK
TITLE =

      A(    ;
      O(    ;
      L     11;
      L     DBW   22;
      ==I   ;
      )     ;
      O(    ;
      L     99;
      L     DBW   22;
      ==I   ;
      )     ;
      )     ;
      FP    DIX   59.2;
      A(    ;
      L     L#0;
      L     DID    0;
      <>D   ;
      )     ;
      =     L     32.0;
      A     L     32.0;
      A(    ;
      L     DBD   24;
      L     DBD    8;
      <>D   ;
      )     ;
      S     DIX   52.0;
      A     L     32.0;
      A(    ;
      L     DBD   24;
      L     DID    0;
      ==D   ;
      )     ;
      A(    ;
      L     DBD   28;
      L     DID    4;
      ==D   ;
      )     ;
      A(    ;
      L     DBD   32;
      L     DID    8;
      ==D   ;
      )     ;
      A(    ;
      L     DBD   36;
      L     DID   12;
      ==D   ;
      )     ;
      S     DIX   52.1;
      A     L     32.0;
      BLD   102;
      S     DIX   61.2;
NETWORK
TITLE =
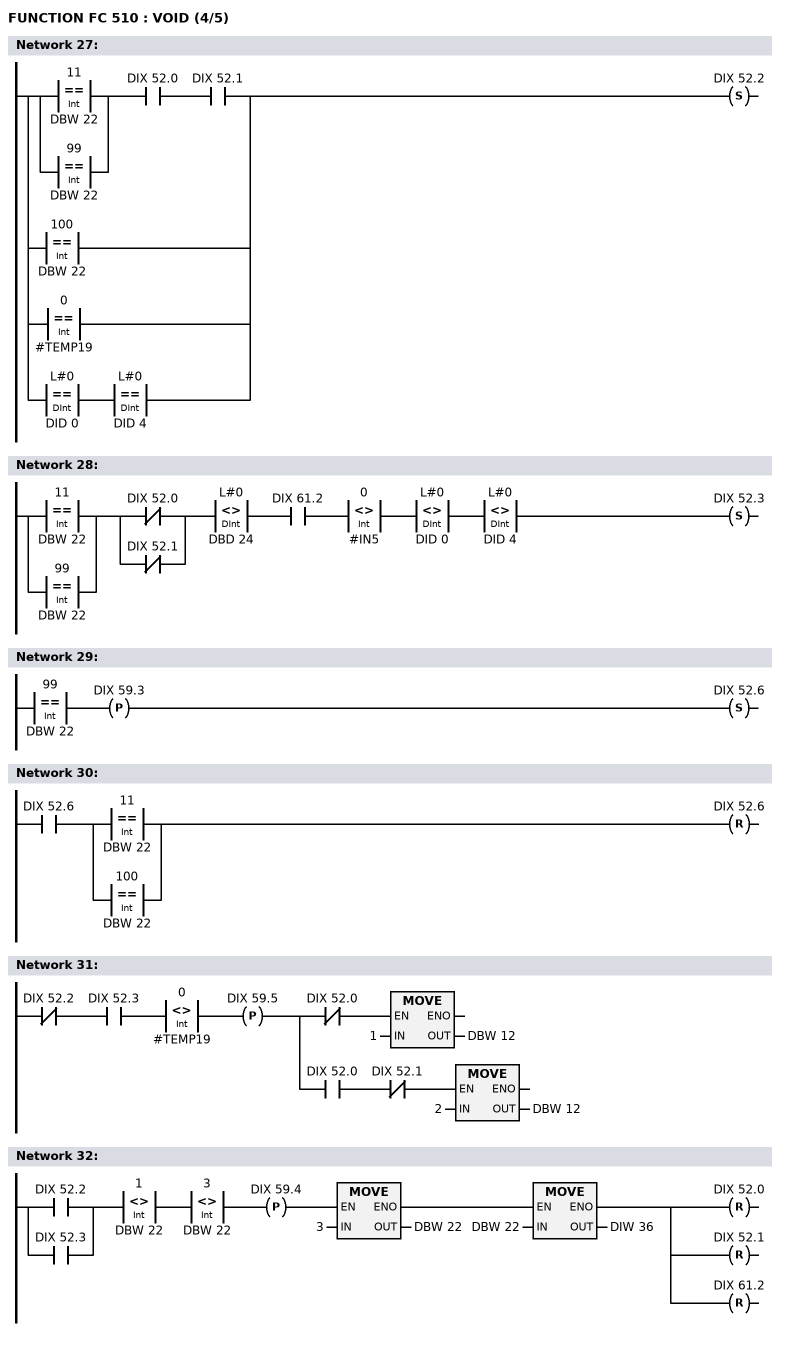

      A(    ;
      O(    ;
      L     11;
      L     DBW   22;
      ==I   ;
      )     ;
      O(    ;
      L     99;
      L     DBW   22;
      ==I   ;
      )     ;
      )     ;
      A     DIX   52.0;
      A     DIX   52.1;
      O(    ;
      L     100;
      L     DBW   22;
      ==I   ;
      )     ;
      O(    ;
      L     0;
      L     #TEMP19;
      ==I   ;
      )     ;
      O     ;
      A(    ;
      L     L#0;
      L     DID    0;
      ==D   ;
      )     ;
      A(    ;
      L     L#0;
      L     DID    4;
      ==D   ;
      )     ;
      S     DIX   52.2;
NETWORK
TITLE =

      A(    ;
      O(    ;
      L     11;
      L     DBW   22;
      ==I   ;
      )     ;
      O(    ;
      L     99;
      L     DBW   22;
      ==I   ;
      )     ;
      )     ;
      A(    ;
      ON    DIX   52.0;
      ON    DIX   52.1;
      )     ;
      A(    ;
      L     L#0;
      L     DBD   24;
      <>D   ;
      )     ;
      A     DIX   61.2;
      A(    ;
      L     0;
      L     #IN5;
      <>I   ;
      )     ;
      A(    ;
      L     L#0;
      L     DID    0;
      <>D   ;
      )     ;
      A(    ;
      L     L#0;
      L     DID    4;
      <>D   ;
      )     ;
      S     DIX   52.3;
NETWORK
TITLE =

      A(    ;
      L     99;
      L     DBW   22;
      ==I   ;
      )     ;
      FP    DIX   59.3;
      S     DIX   52.6;
NETWORK
TITLE =

      A     DIX   52.6;
      A(    ;
      O(    ;
      L     11;
      L     DBW   22;
      ==I   ;
      )     ;
      O(    ;
      L     100;
      L     DBW   22;
      ==I   ;
      )     ;
      )     ;
      R     DIX   52.6;
NETWORK
TITLE =

      AN    DIX   52.2;
      A     DIX   52.3;
      A(    ;
      L     0;
      L     #TEMP19;
      <>I   ;
      )     ;
      FP    DIX   59.5;
      =     L     32.0;
      A     L     32.0;
      AN    DIX   52.0;
      JNB   _01d;
      L     1;
      T     DBW   12;
_01d: NOP   0;
      A     L     32.0;
      A     DIX   52.0;
      AN    DIX   52.1;
      JNB   _01e;
      L     2;
      T     DBW   12;
_01e: NOP   0;
NETWORK
TITLE =

      A(    ;
      A(    ;
      O     DIX   52.2;
      O     DIX   52.3;
      )     ;
      A(    ;
      L     1;
      L     DBW   22;
      <>I   ;
      )     ;
      A(    ;
      L     3;
      L     DBW   22;
      <>I   ;
      )     ;
      FP    DIX   59.4;
      JNB   _01f;
      L     3;
      T     DBW   22;
      SET   ;
      SAVE  ;
      CLR   ;
_01f: A     BR;
      )     ;
      JNB   _020;
      L     DBW   22;
      T     DIW   36;
      SET   ;
      SAVE  ;
      CLR   ;
_020: A     BR;
      R     DIX   52.0;
      R     DIX   52.1;
      R     DIX   61.2;
NETWORK
TITLE =
